LIN {X -0.262,Y -705.428,Z 1161.453,A 0.000,B 0.000,C 90.000,E1 117.462} C_DIS
LIN {X -0.017,Y -706.101,Z 1161.449,A 0.000,B 0.000,C 90.000,E1 116.744} C_DIS
LIN {X 0.213,Y -706.582,Z 1161.443,A 0.000,B 0.000,C 90.000,E1 115.796} C_DIS
LIN {X 0.157,Y -706.745,Z 1161.440,A 0.000,B 0.000,C 90.000,E1 115.103} C_DIS
LIN {X 0.105,Y -706.466,Z 1161.437,A 0.000,B 0.000,C 90.000,E1 114.643} C_DIS
LIN {X 0.398,Y -706.184,Z 1161.436,A 0.000,B 0.000,C 90.000,E1 114.387} C_DIS
LIN {X 0.046,Y -705.311,Z 1161.433,A 0.000,B 0.000,C 90.000,E1 113.951} C_DIS
LIN {X -0.310,Y -703.330,Z 1161.431,A 0.000,B 0.000,C 90.000,E1 113.515} C_DIS
LIN {X -0.028,Y -702.160,Z 1161.429,A 0.000,B 0.000,C 90.000,E1 113.259} C_DIS
LIN {X -0.027,Y -700.058,Z 1161.428,A 0.000,B 0.000,C 90.000,E1 113.025} C_DIS
LIN {X 0.371,Y -696.559,Z 1161.426,A 0.000,B 0.000,C 90.000,E1 112.642} C_DIS
LIN {X -0.143,Y -694.698,Z 1161.425,A 0.000,B 0.000,C 90.000,E1 112.567} C_DIS
LIN {X -0.188,Y -689.270,Z 1161.424,A 0.000,B 0.000,C 90.000,E1 112.386} C_DIS
LIN {X -0.184,Y -686.002,Z 1161.424,A 0.000,B 0.000,C 90.000,E1 112.280} C_DIS
LIN {X -0.175,Y -685.095,Z 1161.424,A 0.000,B 0.000,C 90.000,E1 112.259} C_DIS
LIN {X 0.074,Y -681.362,Z 1161.423,A 0.000,B 0.000,C 90.000,E1 112.206} C_DIS
LIN {X -0.288,Y -676.379,Z 1161.423,A 0.000,B 0.000,C 90.000,E1 112.206} C_DIS
LIN {X 0.256,Y -604.263,Z 1161.423,A 0.000,B 0.000,C 90.000,E1 112.153} C_DIS
LIN {X -0.142,Y -600.886,Z 1161.422,A 0.000,B 0.000,C 90.000,E1 111.972} C_DIS
LIN {X 0.084,Y -595.436,Z 1161.420,A 0.000,B 0.000,C 90.000,E1 111.535} C_DIS
LIN {X -0.058,Y -578.311,Z 1161.411,A 0.000,B 0.000,C 90.000,E1 110.066} C_DIS
LIN {X -0.053,Y -574.045,Z 1161.410,A 0.000,B 0.000,C 90.000,E1 109.704} C_DIS
LIN {X -0.238,Y -568.064,Z 1161.407,A 0.000,B 0.000,C 90.000,E1 109.268} C_DIS
LIN {X -0.148,Y -560.191,Z 1161.404,A 0.000,B 0.000,C 90.000,E1 108.725} C_DIS
LIN {X -0.132,Y -555.536,Z 1161.402,A 0.000,B 0.000,C 90.000,E1 108.417} C_DIS
LIN {X -0.186,Y -551.660,Z 1161.401,A 0.000,B 0.000,C 90.000,E1 108.109} C_DIS
LIN {X 0.019,Y -550.319,Z 1161.399,A 0.000,B 0.000,C 90.000,E1 107.873} C_DIS
LIN {X -0.023,Y -550.302,Z 1161.399,A 0.000,B 0.000,C 90.000,E1 107.873} C_DIS
LIN {X -0.264,Y -550.002,Z 1161.398,A 0.000,B 0.000,C 90.000,E1 107.583} C_DIS
LIN {X -0.119,Y -550.184,Z 1161.394,A 0.000,B 0.000,C 90.000,E1 106.968} C_DIS
LIN {X 0.015,Y -551.315,Z 1161.386,A 0.000,B 0.000,C 90.000,E1 105.552} C_DIS
LIN {X 0.018,Y -552.901,Z 1161.376,A 0.000,B 0.000,C 90.000,E1 103.592} C_DIS
LIN {X -0.071,Y -554.962,Z 1161.363,A 0.000,B 0.000,C 90.000,E1 101.366} C_DIS
LIN {X -0.095,Y -556.105,Z 1161.357,A 0.000,B 0.000,C 90.000,E1 100.254} C_DIS
LIN {X 0.066,Y -557.646,Z 1161.348,A 0.000,B 0.000,C 90.000,E1 98.568} C_DIS
LIN {X 0.038,Y -558.878,Z 1161.340,A 0.000,B 0.000,C 90.000,E1 97.182} C_DIS
LIN {X 0.244,Y -560.316,Z 1161.329,A 0.000,B 0.000,C 90.000,E1 95.220} C_DIS
LIN {X -0.267,Y -561.478,Z 1161.320,A 0.000,B 0.000,C 90.000,E1 93.612} C_DIS
LIN {X -0.219,Y -562.750,Z 1161.311,A 0.000,B 0.000,C 90.000,E1 91.949} C_DIS
LIN {X -0.250,Y -563.791,Z 1161.303,A 0.000,B 0.000,C 90.000,E1 90.573} C_DIS
LIN {X 0.180,Y -564.631,Z 1161.297,A 0.000,B 0.000,C 90.000,E1 89.427} C_DIS
LIN {X -0.271,Y -565.665,Z 1161.288,A 0.000,B 0.000,C 90.000,E1 87.822} C_DIS
LIN {X -0.139,Y -566.641,Z 1161.279,A 0.000,B 0.000,C 90.000,E1 86.159} C_DIS
LIN {X 0.200,Y -567.813,Z 1161.268,A 0.000,B 0.000,C 90.000,E1 84.204} C_DIS
LIN {X -0.212,Y -568.704,Z 1161.260,A 0.000,B 0.000,C 90.000,E1 82.875} C_DIS
LIN {X -0.043,Y -569.488,Z 1161.253,A 0.000,B 0.000,C 90.000,E1 81.489} C_DIS
LIN {X 0.221,Y -570.126,Z 1161.245,A 0.000,B 0.000,C 90.000,E1 80.095} C_DIS
LIN {X 0.122,Y -570.936,Z 1161.236,A 0.000,B 0.000,C 90.000,E1 78.465} C_DIS
LIN {X -0.235,Y -571.445,Z 1161.230,A 0.000,B 0.000,C 90.000,E1 77.409} C_DIS
LIN {X 0.126,Y -572.386,Z 1161.219,A 0.000,B 0.000,C 90.000,E1 75.463} C_DIS
LIN {X -0.259,Y -573.550,Z 1161.207,A 0.000,B 0.000,C 90.000,E1 73.323} C_DIS
LIN {X -0.089,Y -574.421,Z 1161.200,A 0.000,B 0.000,C 90.000,E1 71.945} C_DIS
LIN {X -0.261,Y -576.180,Z 1161.186,A 0.000,B 0.000,C 90.000,E1 69.518} C_DIS
LIN {X -0.193,Y -577.810,Z 1161.176,A 0.000,B 0.000,C 90.000,E1 67.614} C_DIS
LIN {X -0.021,Y -579.444,Z 1161.167,A 0.000,B 0.000,C 90.000,E1 65.973} C_DIS
LIN {X 0.198,Y -580.890,Z 1161.158,A 0.000,B 0.000,C 90.000,E1 64.332} C_DIS
LIN {X -0.215,Y -582.678,Z 1161.147,A 0.000,B 0.000,C 90.000,E1 62.487} C_DIS
LIN {X -0.077,Y -583.908,Z 1161.140,A 0.000,B 0.000,C 90.000,E1 61.129} C_DIS
LIN {X -0.143,Y -585.014,Z 1161.132,A 0.000,B 0.000,C 90.000,E1 59.793} C_DIS
LIN {X -0.357,Y -585.879,Z 1161.126,A 0.000,B 0.000,C 90.000,E1 58.742} C_DIS
LIN {X -0.209,Y -586.962,Z 1161.117,A 0.000,B 0.000,C 90.000,E1 57.120} C_DIS
LIN {X 0.225,Y -587.735,Z 1161.111,A 0.000,B 0.000,C 90.000,E1 56.008} C_DIS
LIN {X 0.251,Y -588.690,Z 1161.102,A 0.000,B 0.000,C 90.000,E1 54.402} C_DIS
LIN {X 0.020,Y -589.819,Z 1161.092,A 0.000,B 0.000,C 90.000,E1 52.557} C_DIS
LIN {X -0.249,Y -590.539,Z 1161.085,A 0.000,B 0.000,C 90.000,E1 51.251} C_DIS
LIN {X 0.115,Y -591.104,Z 1161.079,A 0.000,B 0.000,C 90.000,E1 50.150} C_DIS
LIN {X -0.174,Y -591.386,Z 1161.074,A 0.000,B 0.000,C 90.000,E1 49.380} C_DIS
LIN {X 0.104,Y -591.737,Z 1161.065,A 0.000,B 0.000,C 90.000,E1 47.757} C_DIS
LIN {X -0.213,Y -591.813,Z 1161.058,A 0.000,B 0.000,C 90.000,E1 46.458} C_DIS
LIN {X -0.319,Y -591.679,Z 1161.052,A 0.000,B 0.000,C 90.000,E1 45.405} C_DIS
LIN {X 0.047,Y -591.602,Z 1161.049,A 0.000,B 0.000,C 90.000,E1 44.838} C_DIS
LIN {X -0.062,Y -591.163,Z 1161.043,A 0.000,B 0.000,C 90.000,E1 43.785} C_DIS
LIN {X 0.009,Y -590.467,Z 1161.036,A 0.000,B 0.000,C 90.000,E1 42.447} C_DIS
LIN {X -0.086,Y -589.582,Z 1161.030,A 0.000,B 0.000,C 90.000,E1 41.391} C_DIS
LIN {X 0.010,Y -588.204,Z 1161.023,A 0.000,B 0.000,C 90.000,E1 40.048} C_DIS
LIN {X -0.304,Y -587.257,Z 1161.018,A 0.000,B 0.000,C 90.000,E1 39.277} C_DIS
LIN {X 0.203,Y -585.495,Z 1161.011,A 0.000,B 0.000,C 90.000,E1 37.890} C_DIS
LIN {X -0.328,Y -583.805,Z 1161.005,A 0.000,B 0.000,C 90.000,E1 36.870} C_DIS
LIN {X 0.055,Y -581.695,Z 1160.999,A 0.000,B 0.000,C 90.000,E1 35.758} C_DIS
LIN {X 0.102,Y -579.797,Z 1160.994,A 0.000,B 0.000,C 90.000,E1 34.945} C_DIS
LIN {X 0.264,Y -577.702,Z 1160.990,A 0.000,B 0.000,C 90.000,E1 34.119} C_DIS
LIN {X -0.392,Y -575.196,Z 1160.985,A 0.000,B 0.000,C 90.000,E1 33.372} C_DIS
LIN {X -0.102,Y -573.425,Z 1160.982,A 0.000,B 0.000,C 90.000,E1 32.801} C_DIS
LIN {X 0.295,Y -569.267,Z 1160.976,A 0.000,B 0.000,C 90.000,E1 31.671} C_DIS
LIN {X 0.047,Y -565.634,Z 1160.972,A 0.000,B 0.000,C 90.000,E1 30.875} C_DIS
LIN {X -0.141,Y -562.314,Z 1160.968,A 0.000,B 0.000,C 90.000,E1 30.207} C_DIS
LIN {X 0.195,Y -557.244,Z 1160.962,A 0.000,B 0.000,C 90.000,E1 29.205} C_DIS
LIN {X -0.076,Y -553.266,Z 1160.958,A 0.000,B 0.000,C 90.000,E1 28.537} C_DIS
LIN {X -0.039,Y -549.883,Z 1160.955,A 0.000,B 0.000,C 90.000,E1 27.975} C_DIS
LIN {X 0.231,Y -546.282,Z 1160.952,A 0.000,B 0.000,C 90.000,E1 27.385} C_DIS
LIN {X -0.134,Y -543.457,Z 1160.950,A 0.000,B 0.000,C 90.000,E1 27.001} C_DIS
LIN {X -0.047,Y -538.223,Z 1160.946,A 0.000,B 0.000,C 90.000,E1 26.283} C_DIS
LIN {X -0.107,Y -533.817,Z 1160.943,A 0.000,B 0.000,C 90.000,E1 25.720} C_DIS
LIN {X -0.008,Y -526.846,Z 1160.938,A 0.000,B 0.000,C 90.000,E1 24.847} C_DIS
LIN {X -0.137,Y -519.286,Z 1160.933,A 0.000,B 0.000,C 90.000,E1 24.003} C_DIS
LIN {X 0.240,Y -512.837,Z 1160.929,A 0.000,B 0.000,C 90.000,E1 23.259} C_DIS
LIN {X -0.093,Y -505.969,Z 1160.926,A 0.000,B 0.000,C 90.000,E1 22.589} C_DIS
LIN {X 0.046,Y -500.450,Z 1160.922,A 0.000,B 0.000,C 90.000,E1 22.025} C_DIS
LIN {X -0.062,Y -490.576,Z 1160.917,A 0.000,B 0.000,C 90.000,E1 21.099} C_DIS
LIN {X -0.006,Y -480.430,Z 1160.912,A 0.000,B 0.000,C 90.000,E1 20.174} C_DIS
LIN {X -0.115,Y -467.433,Z 1160.906,A 0.000,B 0.000,C 90.000,E1 19.014} C_DIS
LIN {X 0.017,Y -442.601,Z 1160.893,A 0.000,B 0.000,C 90.000,E1 16.732} C_DIS
LIN {X 0.098,Y -429.624,Z 1160.886,A 0.000,B 0.000,C 90.000,E1 15.426} C_DIS
LIN {X -0.121,Y -416.956,Z 1160.878,A 0.000,B 0.000,C 90.000,E1 14.064} C_DIS
LIN {X -0.221,Y -406.260,Z 1160.871,A 0.000,B 0.000,C 90.000,E1 12.771} C_DIS
LIN {X 0.195,Y -397.899,Z 1160.864,A 0.000,B 0.000,C 90.000,E1 11.535} C_DIS
LIN {X -0.133,Y -395.271,Z 1160.862,A 0.000,B 0.000,C 90.000,E1 11.130} C_DIS
LIN {X 0.077,Y -393.627,Z 1160.860,A 0.000,B 0.000,C 90.000,E1 10.715} C_DIS
LIN {X 0.022,Y -392.924,Z 1160.859,A 0.000,B 0.000,C 90.000,E1 10.546} C_DIS
LIN {X -0.016,Y -392.907,Z 1160.859,A 0.000,B 0.000,C 90.000,E1 10.546} C_DIS
LIN {X 0.149,Y -392.617,Z 1160.856,A 0.000,B 0.000,C 90.000,E1 10.084} C_DIS
LIN {X -0.047,Y -393.292,Z 1160.854,A 0.000,B 0.000,C 90.000,E1 9.670} C_DIS
LIN {X -0.129,Y -395.148,Z 1160.850,A 0.000,B 0.000,C 90.000,E1 8.973} C_DIS
LIN {X 0.162,Y -398.575,Z 1160.844,A 0.000,B 0.000,C 90.000,E1 7.871} C_DIS
LIN {X -0.086,Y -401.754,Z 1160.839,A 0.000,B 0.000,C 90.000,E1 7.068} C_DIS
LIN {X -0.104,Y -405.686,Z 1160.835,A 0.000,B 0.000,C 90.000,E1 6.372} C_DIS
LIN {X -0.128,Y -406.747,Z 1160.834,A 0.000,B 0.000,C 90.000,E1 6.201} C_DIS
LIN {X 0.009,Y -407.934,Z 1160.834,A 0.000,B 0.000,C 90.000,E1 6.030} C_DIS
LIN {X -0.107,Y -410.829,Z 1160.832,A 0.000,B 0.000,C 90.000,E1 5.739} C_DIS
LIN {X -0.033,Y -414.950,Z 1160.830,A 0.000,B 0.000,C 90.000,E1 5.391} C_DIS
LIN {X -0.070,Y -429.560,Z 1160.824,A 0.000,B 0.000,C 90.000,E1 4.302} C_DIS
LIN {X -0.226,Y -444.055,Z 1160.818,A 0.000,B 0.000,C 90.000,E1 3.269} C_DIS
LIN {X 0.022,Y -465.153,Z 1160.810,A 0.000,B 0.000,C 90.000,E1 1.776} C_DIS
LIN {X -0.135,Y -476.141,Z 1160.806,A 0.000,B 0.000,C 90.000,E1 1.031} C_DIS
LIN {X -0.094,Y -483.837,Z 1160.802,A 0.000,B 0.000,C 90.000,E1 0.458} C_DIS
LIN {X 0.000,Y -489.788,Z 1160.800,A 0.000,B 0.000,C 90.000,E1 360.000} C_DIS
LIN {X -0.023,Y -496.862,Z 1160.797,A 0.000,B 0.000,C 90.000,E1 359.427} C_DIS
LIN {X -0.096,Y -504.041,Z 1160.793,A 0.000,B 0.000,C 90.000,E1 358.797} C_DIS
LIN {X 0.239,Y -509.609,Z 1160.790,A 0.000,B 0.000,C 90.000,E1 358.224} C_DIS
LIN {X -0.168,Y -516.066,Z 1160.787,A 0.000,B 0.000,C 90.000,E1 357.593} C_DIS
LIN {X 0.067,Y -522.425,Z 1160.783,A 0.000,B 0.000,C 90.000,E1 356.846} C_DIS
LIN {X 0.244,Y -528.292,Z 1160.779,A 0.000,B 0.000,C 90.000,E1 356.102} C_DIS
LIN {X 0.224,Y -532.626,Z 1160.775,A 0.000,B 0.000,C 90.000,E1 355.527} C_DIS
LIN {X -0.036,Y -537.342,Z 1160.771,A 0.000,B 0.000,C 90.000,E1 354.837} C_DIS
LIN {X -0.257,Y -541.657,Z 1160.767,A 0.000,B 0.000,C 90.000,E1 354.147} C_DIS
LIN {X 0.158,Y -545.578,Z 1160.763,A 0.000,B 0.000,C 90.000,E1 353.394} C_DIS
LIN {X 0.267,Y -548.451,Z 1160.760,A 0.000,B 0.000,C 90.000,E1 352.818} C_DIS
LIN {X 0.247,Y -552.943,Z 1160.755,A 0.000,B 0.000,C 90.000,E1 351.837} C_DIS
LIN {X 0.229,Y -555.790,Z 1160.751,A 0.000,B 0.000,C 90.000,E1 351.141} C_DIS
LIN {X -0.017,Y -558.814,Z 1160.746,A 0.000,B 0.000,C 90.000,E1 350.330} C_DIS
LIN {X -0.137,Y -561.551,Z 1160.742,A 0.000,B 0.000,C 90.000,E1 349.511} C_DIS
LIN {X 0.219,Y -564.082,Z 1160.737,A 0.000,B 0.000,C 90.000,E1 348.645} C_DIS
LIN {X -0.058,Y -567.941,Z 1160.729,A 0.000,B 0.000,C 90.000,E1 347.297} C_DIS
LIN {X -0.139,Y -571.408,Z 1160.722,A 0.000,B 0.000,C 90.000,E1 345.936} C_DIS
LIN {X 0.208,Y -574.072,Z 1160.716,A 0.000,B 0.000,C 90.000,E1 344.810} C_DIS
LIN {X -0.316,Y -577.142,Z 1160.708,A 0.000,B 0.000,C 90.000,E1 343.504} C_DIS
LIN {X 0.307,Y -580.713,Z 1160.699,A 0.000,B 0.000,C 90.000,E1 341.819} C_DIS
LIN {X 0.003,Y -582.324,Z 1160.695,A 0.000,B 0.000,C 90.000,E1 341.040} C_DIS
LIN {X 0.310,Y -584.331,Z 1160.689,A 0.000,B 0.000,C 90.000,E1 339.934} C_DIS
LIN {X 0.312,Y -586.470,Z 1160.681,A 0.000,B 0.000,C 90.000,E1 338.592} C_DIS
LIN {X -0.160,Y -587.244,Z 1160.678,A 0.000,B 0.000,C 90.000,E1 338.103} C_DIS
LIN {X 0.097,Y -588.618,Z 1160.671,A 0.000,B 0.000,C 90.000,E1 336.741} C_DIS
LIN {X 0.294,Y -589.141,Z 1160.666,A 0.000,B 0.000,C 90.000,E1 335.921} C_DIS
LIN {X -0.034,Y -589.396,Z 1160.662,A 0.000,B 0.000,C 90.000,E1 335.153} C_DIS
LIN {X 0.178,Y -589.369,Z 1160.658,A 0.000,B 0.000,C 90.000,E1 334.332} C_DIS
LIN {X -0.142,Y -589.023,Z 1160.653,A 0.000,B 0.000,C 90.000,E1 333.563} C_DIS
LIN {X 0.059,Y -588.261,Z 1160.649,A 0.000,B 0.000,C 90.000,E1 332.743} C_DIS
LIN {X -0.163,Y -587.616,Z 1160.646,A 0.000,B 0.000,C 90.000,E1 332.231} C_DIS
LIN {X -0.228,Y -586.211,Z 1160.641,A 0.000,B 0.000,C 90.000,E1 331.435} C_DIS
LIN {X 0.209,Y -584.479,Z 1160.637,A 0.000,B 0.000,C 90.000,E1 330.589} C_DIS
LIN {X 0.118,Y -582.277,Z 1160.632,A 0.000,B 0.000,C 90.000,E1 329.793} C_DIS
LIN {X 0.004,Y -579.589,Z 1160.628,A 0.000,B 0.000,C 90.000,E1 328.997} C_DIS
LIN {X -0.063,Y -576.929,Z 1160.624,A 0.000,B 0.000,C 90.000,E1 328.329} C_DIS
LIN {X 0.064,Y -572.768,Z 1160.620,A 0.000,B 0.000,C 90.000,E1 327.502} C_DIS
LIN {X 0.023,Y -569.600,Z 1160.617,A 0.000,B 0.000,C 90.000,E1 326.962} C_DIS
LIN {X 0.073,Y -564.104,Z 1160.612,A 0.000,B 0.000,C 90.000,E1 326.135} C_DIS
LIN {X -0.031,Y -560.179,Z 1160.609,A 0.000,B 0.000,C 90.000,E1 325.595} C_DIS
LIN {X -0.050,Y -556.903,Z 1160.607,A 0.000,B 0.000,C 90.000,E1 325.182} C_DIS
LIN {X 0.137,Y -551.314,Z 1160.603,A 0.000,B 0.000,C 90.000,E1 324.482} C_DIS
LIN {X 0.302,Y -543.898,Z 1160.598,A 0.000,B 0.000,C 90.000,E1 323.623} C_DIS
LIN {X -0.197,Y -536.207,Z 1160.594,A 0.000,B 0.000,C 90.000,E1 322.844} C_DIS
LIN {X 0.016,Y -529.985,Z 1160.590,A 0.000,B 0.000,C 90.000,E1 322.145} C_DIS
LIN {X 0.327,Y -527.584,Z 1160.588,A 0.000,B 0.000,C 90.000,E1 321.823} C_DIS
LIN {X 0.268,Y -524.788,Z 1160.586,A 0.000,B 0.000,C 90.000,E1 321.457} C_DIS
LIN {X 0.044,Y -522.012,Z 1160.583,A 0.000,B 0.000,C 90.000,E1 321.009} C_DIS
LIN {X -0.141,Y -521.321,Z 1160.583,A 0.000,B 0.000,C 90.000,E1 320.884} C_DIS
LIN {X -0.227,Y -519.739,Z 1160.580,A 0.000,B 0.000,C 90.000,E1 320.436} C_DIS
LIN {X 0.132,Y -518.543,Z 1160.576,A 0.000,B 0.000,C 90.000,E1 319.666} C_DIS
LIN {X -0.033,Y -518.632,Z 1160.569,A 0.000,B 0.000,C 90.000,E1 318.366} C_DIS
LIN {X -0.127,Y -519.406,Z 1160.559,A 0.000,B 0.000,C 90.000,E1 316.620} C_DIS
LIN {X 0.045,Y -520.418,Z 1160.548,A 0.000,B 0.000,C 90.000,E1 314.555} C_DIS
LIN {X -0.051,Y -521.275,Z 1160.538,A 0.000,B 0.000,C 90.000,E1 312.813} C_DIS
LIN {X -0.143,Y -522.416,Z 1160.526,A 0.000,B 0.000,C 90.000,E1 310.782} C_DIS
LIN {X -0.197,Y -523.548,Z 1160.515,A 0.000,B 0.000,C 90.000,E1 308.749} C_DIS
LIN {X -0.116,Y -524.617,Z 1160.505,A 0.000,B 0.000,C 90.000,E1 306.996} C_DIS
LIN {X 0.162,Y -525.317,Z 1160.499,A 0.000,B 0.000,C 90.000,E1 305.804} C_DIS
LIN {X -0.311,Y -526.137,Z 1160.491,A 0.000,B 0.000,C 90.000,E1 304.405} C_DIS
LIN {X 0.002,Y -527.633,Z 1160.478,A 0.000,B 0.000,C 90.000,E1 302.054} C_DIS
LIN {X -0.142,Y -528.689,Z 1160.469,A 0.000,B 0.000,C 90.000,E1 300.335} C_DIS
LIN {X -0.070,Y -529.202,Z 1160.464,A 0.000,B 0.000,C 90.000,E1 299.461} C_DIS
LIN {X -0.090,Y -529.711,Z 1160.457,A 0.000,B 0.000,C 90.000,E1 298.309} C_DIS
LIN {X -0.021,Y -530.066,Z 1160.453,A 0.000,B 0.000,C 90.000,E1 297.436} C_DIS
LIN {X -0.142,Y -530.367,Z 1160.443,A 0.000,B 0.000,C 90.000,E1 295.720} C_DIS
LIN {X 0.041,Y -530.419,Z 1160.435,A 0.000,B 0.000,C 90.000,E1 294.259} C_DIS
LIN {X -0.113,Y -530.369,Z 1160.424,A 0.000,B 0.000,C 90.000,E1 292.259} C_DIS
LIN {X 0.138,Y -530.298,Z 1160.416,A 0.000,B 0.000,C 90.000,E1 290.791} C_DIS
LIN {X -0.101,Y -529.831,Z 1160.406,A 0.000,B 0.000,C 90.000,E1 289.087} C_DIS
LIN {X -0.210,Y -529.453,Z 1160.400,A 0.000,B 0.000,C 90.000,E1 287.946} C_DIS
LIN {X -0.128,Y -528.736,Z 1160.390,A 0.000,B 0.000,C 90.000,E1 286.205} C_DIS
LIN {X 0.088,Y -528.396,Z 1160.385,A 0.000,B 0.000,C 90.000,E1 285.315} C_DIS
LIN {X -0.006,Y -527.467,Z 1160.376,A 0.000,B 0.000,C 90.000,E1 283.592} C_DIS
LIN {X 0.210,Y -526.778,Z 1160.369,A 0.000,B 0.000,C 90.000,E1 282.411} C_DIS
LIN {X -0.195,Y -525.859,Z 1160.361,A 0.000,B 0.000,C 90.000,E1 281.007} C_DIS
LIN {X -0.193,Y -524.860,Z 1160.353,A 0.000,B 0.000,C 90.000,E1 279.557} C_DIS
LIN {X -0.195,Y -523.779,Z 1160.343,A 0.000,B 0.000,C 90.000,E1 277.814} C_DIS
LIN {X 0.161,Y -522.723,Z 1160.334,A 0.000,B 0.000,C 90.000,E1 276.030} C_DIS
LIN {X -0.017,Y -521.895,Z 1160.324,A 0.000,B 0.000,C 90.000,E1 274.302} C_DIS
LIN {X -0.209,Y -521.260,Z 1160.316,A 0.000,B 0.000,C 90.000,E1 272.865} C_DIS
LIN {X 0.077,Y -520.691,Z 1160.308,A 0.000,B 0.000,C 90.000,E1 271.375} C_DIS
LIN {X -0.178,Y -520.061,Z 1160.300,A 0.000,B 0.000,C 90.000,E1 269.943} C_DIS
LIN {X 0.074,Y -519.452,Z 1160.292,A 0.000,B 0.000,C 90.000,E1 268.453} C_DIS
LIN {X -0.195,Y -518.750,Z 1160.283,A 0.000,B 0.000,C 90.000,E1 267.020} C_DIS
LIN {X 0.072,Y -517.852,Z 1160.275,A 0.000,B 0.000,C 90.000,E1 265.527} C_DIS
LIN {X -0.194,Y -516.745,Z 1160.267,A 0.000,B 0.000,C 90.000,E1 264.090} C_DIS
LIN {X 0.058,Y -515.023,Z 1160.257,A 0.000,B 0.000,C 90.000,E1 262.299} C_DIS
LIN {X -0.158,Y -513.287,Z 1160.247,A 0.000,B 0.000,C 90.000,E1 260.557} C_DIS
LIN {X 0.060,Y -511.322,Z 1160.236,A 0.000,B 0.000,C 90.000,E1 258.465} C_DIS
LIN {X -0.118,Y -509.260,Z 1160.223,A 0.000,B 0.000,C 90.000,E1 256.117} C_DIS
LIN {X -0.053,Y -507.467,Z 1160.211,A 0.000,B 0.000,C 90.000,E1 254.031} C_DIS
LIN {X 0.033,Y -505.854,Z 1160.201,A 0.000,B 0.000,C 90.000,E1 252.236} C_DIS
LIN {X 0.231,Y -504.171,Z 1160.191,A 0.000,B 0.000,C 90.000,E1 250.423} C_DIS
LIN {X 0.168,Y -502.118,Z 1160.180,A 0.000,B 0.000,C 90.000,E1 248.337} C_DIS
LIN {X -0.177,Y -500.917,Z 1160.173,A 0.000,B 0.000,C 90.000,E1 247.177} C_DIS
LIN {X 0.236,Y -499.874,Z 1160.168,A 0.000,B 0.000,C 90.000,E1 246.230} C_DIS
LIN {X 0.314,Y -498.049,Z 1160.160,A 0.000,B 0.000,C 90.000,E1 244.717} C_DIS
LIN {X -0.095,Y -496.048,Z 1160.151,A 0.000,B 0.000,C 90.000,E1 243.256} C_DIS
LIN {X 0.118,Y -493.945,Z 1160.143,A 0.000,B 0.000,C 90.000,E1 241.719} C_DIS
LIN {X -0.083,Y -491.277,Z 1160.133,A 0.000,B 0.000,C 90.000,E1 239.921} C_DIS
LIN {X 0.261,Y -489.514,Z 1160.126,A 0.000,B 0.000,C 90.000,E1 238.663} C_DIS
LIN {X -0.014,Y -487.185,Z 1160.118,A 0.000,B 0.000,C 90.000,E1 237.168} C_DIS
LIN {X -0.061,Y -484.884,Z 1160.109,A 0.000,B 0.000,C 90.000,E1 235.642} C_DIS
LIN {X 0.056,Y -482.159,Z 1160.099,A 0.000,B 0.000,C 90.000,E1 233.783} C_DIS
LIN {X -0.012,Y -480.267,Z 1160.092,A 0.000,B 0.000,C 90.000,E1 232.557} C_DIS
LIN {X 0.061,Y -476.440,Z 1160.078,A 0.000,B 0.000,C 90.000,E1 230.070} C_DIS
LIN {X -0.060,Y -474.104,Z 1160.070,A 0.000,B 0.000,C 90.000,E1 228.528} C_DIS
LIN {X 0.126,Y -471.588,Z 1160.061,A 0.000,B 0.000,C 90.000,E1 226.944} C_DIS
LIN {X 0.098,Y -465.961,Z 1160.040,A 0.000,B 0.000,C 90.000,E1 223.176} C_DIS
LIN {X 0.002,Y -462.302,Z 1160.017,A 0.000,B 0.000,C 90.000,E1 219.072} C_DIS
LIN {X -0.181,Y -461.000,Z 1160.005,A 0.000,B 0.000,C 90.000,E1 216.870} C_DIS
LIN {X -0.011,Y -459.562,Z 1159.976,A 0.000,B 0.000,C 90.000,E1 211.750} C_DIS
LIN {X 0.092,Y -460.857,Z 1159.957,A 0.000,B 0.000,C 90.000,E1 208.231} C_DIS
LIN {X -0.214,Y -462.289,Z 1159.946,A 0.000,B 0.000,C 90.000,E1 206.360} C_DIS
LIN {X 0.205,Y -465.295,Z 1159.932,A 0.000,B 0.000,C 90.000,E1 203.770} C_DIS
LIN {X 0.224,Y -471.462,Z 1159.913,A 0.000,B 0.000,C 90.000,E1 200.301} C_DIS
LIN {X 0.082,Y -477.505,Z 1159.899,A 0.000,B 0.000,C 90.000,E1 197.819} C_DIS
LIN {X -0.155,Y -484.717,Z 1159.885,A 0.000,B 0.000,C 90.000,E1 195.371} C_DIS
LIN {X -0.197,Y -490.749,Z 1159.875,A 0.000,B 0.000,C 90.000,E1 193.536} C_DIS
LIN {X -0.127,Y -495.808,Z 1159.867,A 0.000,B 0.000,C 90.000,E1 192.007} C_DIS
LIN {X -0.134,Y -502.173,Z 1159.857,A 0.000,B 0.000,C 90.000,E1 190.197} C_DIS
LIN {X -0.183,Y -510.885,Z 1159.843,A 0.000,B 0.000,C 90.000,E1 187.814} C_DIS
LIN {X 0.008,Y -516.405,Z 1159.835,A 0.000,B 0.000,C 90.000,E1 186.315} C_DIS
LIN {X 0.244,Y -522.816,Z 1159.825,A 0.000,B 0.000,C 90.000,E1 184.531} C_DIS
LIN {X 0.095,Y -527.125,Z 1159.819,A 0.000,B 0.000,C 90.000,E1 183.383} C_DIS
LIN {X -0.006,Y -532.466,Z 1159.811,A 0.000,B 0.000,C 90.000,E1 181.949} C_DIS
LIN {X -0.015,Y -537.760,Z 1159.803,A 0.000,B 0.000,C 90.000,E1 180.516} C_DIS
LIN {X 0.087,Y -544.151,Z 1159.793,A 0.000,B 0.000,C 90.000,E1 178.797} C_DIS
LIN {X -0.211,Y -550.558,Z 1159.784,A 0.000,B 0.000,C 90.000,E1 177.135} C_DIS
LIN {X -0.234,Y -557.962,Z 1159.773,A 0.000,B 0.000,C 90.000,E1 175.179} C_DIS
LIN {X 0.260,Y -563.175,Z 1159.765,A 0.000,B 0.000,C 90.000,E1 173.742} C_DIS
LIN {X -0.120,Y -569.471,Z 1159.756,A 0.000,B 0.000,C 90.000,E1 172.129} C_DIS
LIN {X -0.211,Y -575.692,Z 1159.747,A 0.000,B 0.000,C 90.000,E1 170.500} C_DIS
LIN {X -0.163,Y -581.770,Z 1159.738,A 0.000,B 0.000,C 90.000,E1 168.870} C_DIS
LIN {X 0.207,Y -585.764,Z 1159.732,A 0.000,B 0.000,C 90.000,E1 167.757} C_DIS
LIN {X -0.254,Y -590.583,Z 1159.725,A 0.000,B 0.000,C 90.000,E1 166.464} C_DIS
LIN {X 0.082,Y -595.199,Z 1159.717,A 0.000,B 0.000,C 90.000,E1 165.102} C_DIS
LIN {X 0.047,Y -598.842,Z 1159.711,A 0.000,B 0.000,C 90.000,E1 164.047} C_DIS
LIN {X -0.185,Y -602.353,Z 1159.706,A 0.000,B 0.000,C 90.000,E1 163.015} C_DIS
LIN {X -0.052,Y -606.543,Z 1159.698,A 0.000,B 0.000,C 90.000,E1 161.692} C_DIS
LIN {X 0.088,Y -611.258,Z 1159.690,A 0.000,B 0.000,C 90.000,E1 160.115} C_DIS
LIN {X -0.260,Y -615.792,Z 1159.681,A 0.000,B 0.000,C 90.000,E1 158.592} C_DIS
LIN {X -0.304,Y -620.038,Z 1159.672,A 0.000,B 0.000,C 90.000,E1 157.050} C_DIS
LIN {X -0.023,Y -623.514,Z 1159.665,A 0.000,B 0.000,C 90.000,E1 155.741} C_DIS
LIN {X 0.028,Y -627.493,Z 1159.657,A 0.000,B 0.000,C 90.000,E1 154.204} C_DIS
LIN {X 0.172,Y -631.334,Z 1159.648,A 0.000,B 0.000,C 90.000,E1 152.666} C_DIS
LIN {X 0.308,Y -633.801,Z 1159.643,A 0.000,B 0.000,C 90.000,E1 151.641} C_DIS
LIN {X -0.049,Y -636.689,Z 1159.636,A 0.000,B 0.000,C 90.000,E1 150.411} C_DIS
LIN {X -0.099,Y -638.966,Z 1159.630,A 0.000,B 0.000,C 90.000,E1 149.410} C_DIS
LIN {X -0.117,Y -641.027,Z 1159.625,A 0.000,B 0.000,C 90.000,E1 148.408} C_DIS
LIN {X 0.288,Y -643.463,Z 1159.618,A 0.000,B 0.000,C 90.000,E1 147.120} C_DIS
LIN {X 0.195,Y -645.797,Z 1159.611,A 0.000,B 0.000,C 90.000,E1 145.881} C_DIS
LIN {X 0.136,Y -647.982,Z 1159.604,A 0.000,B 0.000,C 90.000,E1 144.642} C_DIS
LIN {X -0.040,Y -650.110,Z 1159.597,A 0.000,B 0.000,C 90.000,E1 143.417} C_DIS
LIN {X -0.260,Y -653.420,Z 1159.586,A 0.000,B 0.000,C 90.000,E1 141.457} C_DIS
LIN {X 0.016,Y -657.097,Z 1159.575,A 0.000,B 0.000,C 90.000,E1 139.461} C_DIS
LIN {X -0.147,Y -660.626,Z 1159.565,A 0.000,B 0.000,C 90.000,E1 137.757} C_DIS
LIN {X -0.219,Y -663.632,Z 1159.557,A 0.000,B 0.000,C 90.000,E1 136.296} C_DIS
LIN {X -0.253,Y -668.791,Z 1159.544,A 0.000,B 0.000,C 90.000,E1 133.866} C_DIS
LIN {X -0.133,Y -673.295,Z 1159.533,A 0.000,B 0.000,C 90.000,E1 131.919} C_DIS
LIN {X 0.197,Y -678.478,Z 1159.521,A 0.000,B 0.000,C 90.000,E1 129.725} C_DIS
LIN {X 0.002,Y -681.542,Z 1159.514,A 0.000,B 0.000,C 90.000,E1 128.543} C_DIS
LIN {X -0.151,Y -684.520,Z 1159.508,A 0.000,B 0.000,C 90.000,E1 127.363} C_DIS
LIN {X -0.126,Y -687.507,Z 1159.501,A 0.000,B 0.000,C 90.000,E1 126.171} C_DIS
LIN {X -0.011,Y -691.004,Z 1159.493,A 0.000,B 0.000,C 90.000,E1 124.739} C_DIS
LIN {X 0.086,Y -693.272,Z 1159.488,A 0.000,B 0.000,C 90.000,E1 123.785} C_DIS
LIN {X -0.105,Y -696.493,Z 1159.480,A 0.000,B 0.000,C 90.000,E1 122.388} C_DIS
LIN {X 0.035,Y -697.969,Z 1159.476,A 0.000,B 0.000,C 90.000,E1 121.671} C_DIS
LIN {X -0.121,Y -700.212,Z 1159.469,A 0.000,B 0.000,C 90.000,E1 120.512} C_DIS
LIN {X 0.274,Y -702.683,Z 1159.462,A 0.000,B 0.000,C 90.000,E1 119.077} C_DIS
LIN {X 0.157,Y -704.340,Z 1159.457,A 0.000,B 0.000,C 90.000,E1 118.153} C_DIS
LIN {X 0.064,Y -705.376,Z 1159.453,A 0.000,B 0.000,C 90.000,E1 117.462} C_DIS
LIN {X 0.308,Y -706.055,Z 1159.449,A 0.000,B 0.000,C 90.000,E1 116.744} C_DIS
LIN {X -0.099,Y -706.543,Z 1159.444,A 0.000,B 0.000,C 90.000,E1 115.848} C_DIS
LIN {X -0.158,Y -706.735,Z 1159.440,A 0.000,B 0.000,C 90.000,E1 115.155} C_DIS
LIN {X -0.212,Y -706.481,Z 1159.437,A 0.000,B 0.000,C 90.000,E1 114.695} C_DIS
LIN {X -0.213,Y -706.228,Z 1159.436,A 0.000,B 0.000,C 90.000,E1 114.463} C_DIS
LIN {X 0.370,Y -705.358,Z 1159.433,A 0.000,B 0.000,C 90.000,E1 113.951} C_DIS
LIN {X -0.273,Y -704.507,Z 1159.432,A 0.000,B 0.000,C 90.000,E1 113.770} C_DIS
LIN {X 0.295,Y -702.331,Z 1159.429,A 0.000,B 0.000,C 90.000,E1 113.259} C_DIS
LIN {X 0.157,Y -701.438,Z 1159.429,A 0.000,B 0.000,C 90.000,E1 113.153} C_DIS
LIN {X 0.050,Y -696.897,Z 1159.426,A 0.000,B 0.000,C 90.000,E1 112.695} C_DIS
LIN {X -0.088,Y -695.236,Z 1159.426,A 0.000,B 0.000,C 90.000,E1 112.589} C_DIS
LIN {X 0.264,Y -692.820,Z 1159.425,A 0.000,B 0.000,C 90.000,E1 112.461} C_DIS
LIN {X -0.081,Y -685.622,Z 1159.424,A 0.000,B 0.000,C 90.000,E1 112.259} C_DIS
LIN {X 0.167,Y -683.209,Z 1159.423,A 0.000,B 0.000,C 90.000,E1 112.206} C_DIS
LIN {X -0.303,Y -677.072,Z 1159.423,A 0.000,B 0.000,C 90.000,E1 112.206} C_DIS
LIN {X 0.242,Y -604.198,Z 1159.423,A 0.000,B 0.000,C 90.000,E1 112.153} C_DIS
LIN {X -0.070,Y -600.945,Z 1159.422,A 0.000,B 0.000,C 90.000,E1 111.972} C_DIS
LIN {X 0.156,Y -595.490,Z 1159.420,A 0.000,B 0.000,C 90.000,E1 111.535} C_DIS
LIN {X 0.108,Y -578.472,Z 1159.412,A 0.000,B 0.000,C 90.000,E1 110.066} C_DIS
LIN {X 0.112,Y -574.275,Z 1159.410,A 0.000,B 0.000,C 90.000,E1 109.704} C_DIS
LIN {X -0.109,Y -568.255,Z 1159.407,A 0.000,B 0.000,C 90.000,E1 109.268} C_DIS
LIN {X -0.027,Y -560.355,Z 1159.404,A 0.000,B 0.000,C 90.000,E1 108.725} C_DIS
LIN {X -0.010,Y -555.662,Z 1159.402,A 0.000,B 0.000,C 90.000,E1 108.417} C_DIS
LIN {X 0.117,Y -551.453,Z 1159.400,A 0.000,B 0.000,C 90.000,E1 108.055} C_DIS
LIN {X -0.035,Y -550.249,Z 1159.399,A 0.000,B 0.000,C 90.000,E1 107.873} C_DIS
LIN {X -0.077,Y -550.244,Z 1159.399,A 0.000,B 0.000,C 90.000,E1 107.873} C_DIS
LIN {X -0.233,Y -549.962,Z 1159.398,A 0.000,B 0.000,C 90.000,E1 107.583} C_DIS
LIN {X -0.180,Y -550.398,Z 1159.393,A 0.000,B 0.000,C 90.000,E1 106.677} C_DIS
LIN {X 0.220,Y -551.723,Z 1159.383,A 0.000,B 0.000,C 90.000,E1 104.954} C_DIS
LIN {X 0.097,Y -553.331,Z 1159.372,A 0.000,B 0.000,C 90.000,E1 103.008} C_DIS
LIN {X 0.027,Y -555.498,Z 1159.360,A 0.000,B 0.000,C 90.000,E1 100.782} C_DIS
LIN {X 0.006,Y -556.533,Z 1159.354,A 0.000,B 0.000,C 90.000,E1 99.670} C_DIS
LIN {X 0.036,Y -557.829,Z 1159.346,A 0.000,B 0.000,C 90.000,E1 98.276} C_DIS
LIN {X 0.006,Y -559.005,Z 1159.338,A 0.000,B 0.000,C 90.000,E1 96.891} C_DIS
LIN {X 0.074,Y -560.238,Z 1159.329,A 0.000,B 0.000,C 90.000,E1 95.220} C_DIS
LIN {X 0.216,Y -561.625,Z 1159.318,A 0.000,B 0.000,C 90.000,E1 93.269} C_DIS
LIN {X -0.171,Y -563.139,Z 1159.308,A 0.000,B 0.000,C 90.000,E1 91.375} C_DIS
LIN {X 0.005,Y -564.576,Z 1159.297,A 0.000,B 0.000,C 90.000,E1 89.427} C_DIS
LIN {X 0.117,Y -565.591,Z 1159.288,A 0.000,B 0.000,C 90.000,E1 87.764} C_DIS
LIN {X 0.138,Y -566.426,Z 1159.280,A 0.000,B 0.000,C 90.000,E1 86.388} C_DIS
LIN {X -0.089,Y -567.544,Z 1159.269,A 0.000,B 0.000,C 90.000,E1 84.489} C_DIS
LIN {X -0.002,Y -568.424,Z 1159.262,A 0.000,B 0.000,C 90.000,E1 83.109} C_DIS
LIN {X -0.228,Y -569.365,Z 1159.253,A 0.000,B 0.000,C 90.000,E1 81.489} C_DIS
LIN {X 0.220,Y -570.111,Z 1159.244,A 0.000,B 0.000,C 90.000,E1 79.803} C_DIS
LIN {X 0.120,Y -570.933,Z 1159.234,A 0.000,B 0.000,C 90.000,E1 78.173} C_DIS
LIN {X 0.142,Y -571.696,Z 1159.225,A 0.000,B 0.000,C 90.000,E1 76.533} C_DIS
LIN {X -0.245,Y -572.499,Z 1159.216,A 0.000,B 0.000,C 90.000,E1 74.936} C_DIS
LIN {X 0.077,Y -573.744,Z 1159.204,A 0.000,B 0.000,C 90.000,E1 72.725} C_DIS
LIN {X -0.293,Y -574.296,Z 1159.200,A 0.000,B 0.000,C 90.000,E1 71.945} C_DIS
LIN {X 0.273,Y -576.059,Z 1159.186,A 0.000,B 0.000,C 90.000,E1 69.444} C_DIS
LIN {X -0.185,Y -577.694,Z 1159.175,A 0.000,B 0.000,C 90.000,E1 67.592} C_DIS
LIN {X 0.293,Y -579.335,Z 1159.166,A 0.000,B 0.000,C 90.000,E1 65.921} C_DIS
LIN {X -0.155,Y -581.020,Z 1159.156,A 0.000,B 0.000,C 90.000,E1 64.076} C_DIS
LIN {X -0.303,Y -582.328,Z 1159.148,A 0.000,B 0.000,C 90.000,E1 62.743} C_DIS
LIN {X -0.170,Y -583.569,Z 1159.141,A 0.000,B 0.000,C 90.000,E1 61.385} C_DIS
LIN {X 0.265,Y -584.715,Z 1159.134,A 0.000,B 0.000,C 90.000,E1 59.999} C_DIS
LIN {X 0.219,Y -585.744,Z 1159.126,A 0.000,B 0.000,C 90.000,E1 58.663} C_DIS
LIN {X 0.370,Y -586.801,Z 1159.117,A 0.000,B 0.000,C 90.000,E1 57.041} C_DIS
LIN {X -0.009,Y -587.563,Z 1159.111,A 0.000,B 0.000,C 90.000,E1 56.008} C_DIS
LIN {X 0.013,Y -588.519,Z 1159.102,A 0.000,B 0.000,C 90.000,E1 54.402} C_DIS
LIN {X -0.020,Y -589.778,Z 1159.090,A 0.000,B 0.000,C 90.000,E1 52.271} C_DIS
LIN {X 0.335,Y -590.347,Z 1159.084,A 0.000,B 0.000,C 90.000,E1 51.170} C_DIS
LIN {X 0.068,Y -590.977,Z 1159.077,A 0.000,B 0.000,C 90.000,E1 49.865} C_DIS
LIN {X 0.368,Y -591.258,Z 1159.071,A 0.000,B 0.000,C 90.000,E1 48.771} C_DIS
LIN {X -0.152,Y -591.481,Z 1159.065,A 0.000,B 0.000,C 90.000,E1 47.757} C_DIS
LIN {X -0.066,Y -591.546,Z 1159.058,A 0.000,B 0.000,C 90.000,E1 46.419} C_DIS
LIN {X 0.017,Y -591.379,Z 1159.051,A 0.000,B 0.000,C 90.000,E1 45.081} C_DIS
LIN {X -0.094,Y -591.041,Z 1159.045,A 0.000,B 0.000,C 90.000,E1 44.028} C_DIS
LIN {X 0.216,Y -590.427,Z 1159.039,A 0.000,B 0.000,C 90.000,E1 42.933} C_DIS
LIN {X -0.266,Y -590.145,Z 1159.036,A 0.000,B 0.000,C 90.000,E1 42.447} C_DIS
LIN {X 0.024,Y -589.220,Z 1159.030,A 0.000,B 0.000,C 90.000,E1 41.353} C_DIS
LIN {X 0.104,Y -587.825,Z 1159.022,A 0.000,B 0.000,C 90.000,E1 40.011} C_DIS
LIN {X 0.234,Y -586.868,Z 1159.018,A 0.000,B 0.000,C 90.000,E1 39.197} C_DIS
LIN {X -0.090,Y -585.067,Z 1159.010,A 0.000,B 0.000,C 90.000,E1 37.890} C_DIS
LIN {X 0.190,Y -583.384,Z 1159.005,A 0.000,B 0.000,C 90.000,E1 36.790} C_DIS
LIN {X -0.073,Y -580.634,Z 1158.997,A 0.000,B 0.000,C 90.000,E1 35.471} C_DIS
LIN {X -0.043,Y -578.597,Z 1158.993,A 0.000,B 0.000,C 90.000,E1 34.659} C_DIS
LIN {X -0.049,Y -577.156,Z 1158.990,A 0.000,B 0.000,C 90.000,E1 34.119} C_DIS
LIN {X 0.088,Y -574.601,Z 1158.985,A 0.000,B 0.000,C 90.000,E1 33.293} C_DIS
LIN {X 0.060,Y -572.763,Z 1158.982,A 0.000,B 0.000,C 90.000,E1 32.752} C_DIS
LIN {X -0.033,Y -568.592,Z 1158.976,A 0.000,B 0.000,C 90.000,E1 31.671} C_DIS
LIN {X 0.002,Y -564.883,Z 1158.971,A 0.000,B 0.000,C 90.000,E1 30.846} C_DIS
LIN {X 0.102,Y -562.246,Z 1158.968,A 0.000,B 0.000,C 90.000,E1 30.285} C_DIS
LIN {X -0.049,Y -557.184,Z 1158.963,A 0.000,B 0.000,C 90.000,E1 29.333} C_DIS
LIN {X 0.170,Y -553.278,Z 1158.959,A 0.000,B 0.000,C 90.000,E1 28.615} C_DIS
LIN {X 0.090,Y -549.002,Z 1158.955,A 0.000,B 0.000,C 90.000,E1 27.924} C_DIS
LIN {X -0.128,Y -545.345,Z 1158.952,A 0.000,B 0.000,C 90.000,E1 27.385} C_DIS
LIN {X 0.106,Y -541.411,Z 1158.949,A 0.000,B 0.000,C 90.000,E1 26.796} C_DIS
LIN {X -0.067,Y -536.135,Z 1158.945,A 0.000,B 0.000,C 90.000,E1 26.104} C_DIS
LIN {X -0.281,Y -530.506,Z 1158.941,A 0.000,B 0.000,C 90.000,E1 25.412} C_DIS
LIN {X 0.160,Y -524.472,Z 1158.937,A 0.000,B 0.000,C 90.000,E1 24.643} C_DIS
LIN {X -0.212,Y -516.854,Z 1158.932,A 0.000,B 0.000,C 90.000,E1 23.823} C_DIS
LIN {X 0.051,Y -510.071,Z 1158.928,A 0.000,B 0.000,C 90.000,E1 23.078} C_DIS
LIN {X -0.108,Y -501.850,Z 1158.924,A 0.000,B 0.000,C 90.000,E1 22.259} C_DIS
LIN {X 0.215,Y -493.292,Z 1158.919,A 0.000,B 0.000,C 90.000,E1 21.408} C_DIS
LIN {X -0.158,Y -487.547,Z 1158.916,A 0.000,B 0.000,C 90.000,E1 20.918} C_DIS
LIN {X -0.140,Y -477.341,Z 1158.911,A 0.000,B 0.000,C 90.000,E1 19.993} C_DIS
LIN {X 0.187,Y -465.726,Z 1158.905,A 0.000,B 0.000,C 90.000,E1 18.906} C_DIS
LIN {X 0.034,Y -449.398,Z 1158.897,A 0.000,B 0.000,C 90.000,E1 17.457} C_DIS
LIN {X -0.183,Y -431.968,Z 1158.888,A 0.000,B 0.000,C 90.000,E1 15.788} C_DIS
LIN {X -0.143,Y -419.297,Z 1158.880,A 0.000,B 0.000,C 90.000,E1 14.411} C_DIS
LIN {X 0.166,Y -408.346,Z 1158.873,A 0.000,B 0.000,C 90.000,E1 13.063} C_DIS
LIN {X -0.098,Y -400.700,Z 1158.867,A 0.000,B 0.000,C 90.000,E1 12.063} C_DIS
LIN {X -0.072,Y -397.244,Z 1158.864,A 0.000,B 0.000,C 90.000,E1 11.535} C_DIS
LIN {X -0.069,Y -394.328,Z 1158.861,A 0.000,B 0.000,C 90.000,E1 11.007} C_DIS
LIN {X -0.076,Y -392.810,Z 1158.859,A 0.000,B 0.000,C 90.000,E1 10.602} C_DIS
LIN {X -0.185,Y -392.541,Z 1158.857,A 0.000,B 0.000,C 90.000,E1 10.197} C_DIS
LIN {X -0.050,Y -393.541,Z 1158.853,A 0.000,B 0.000,C 90.000,E1 9.557} C_DIS
LIN {X -0.118,Y -396.058,Z 1158.848,A 0.000,B 0.000,C 90.000,E1 8.681} C_DIS
LIN {X 0.147,Y -400.327,Z 1158.841,A 0.000,B 0.000,C 90.000,E1 7.409} C_DIS
LIN {X 0.080,Y -401.637,Z 1158.839,A 0.000,B 0.000,C 90.000,E1 7.068} C_DIS
LIN {X 0.115,Y -403.670,Z 1158.837,A 0.000,B 0.000,C 90.000,E1 6.663} C_DIS
LIN {X -0.196,Y -406.597,Z 1158.834,A 0.000,B 0.000,C 90.000,E1 6.201} C_DIS
LIN {X -0.175,Y -407.917,Z 1158.833,A 0.000,B 0.000,C 90.000,E1 6.024} C_DIS
LIN {X -0.149,Y -411.100,Z 1158.832,A 0.000,B 0.000,C 90.000,E1 5.682} C_DIS
LIN {X 0.002,Y -415.058,Z 1158.830,A 0.000,B 0.000,C 90.000,E1 5.334} C_DIS
LIN {X -0.083,Y -434.515,Z 1158.822,A 0.000,B 0.000,C 90.000,E1 3.898} C_DIS
LIN {X -0.094,Y -457.128,Z 1158.813,A 0.000,B 0.000,C 90.000,E1 2.293} C_DIS
LIN {X -0.201,Y -471.651,Z 1158.807,A 0.000,B 0.000,C 90.000,E1 1.318} C_DIS
LIN {X -0.068,Y -477.954,Z 1158.805,A 0.000,B 0.000,C 90.000,E1 0.859} C_DIS
LIN {X 0.000,Y -489.349,Z 1158.800,A 0.000,B 0.000,C 90.000,E1 360.000} C_DIS
LIN {X 0.009,Y -496.489,Z 1158.797,A 0.000,B 0.000,C 90.000,E1 359.427} C_DIS
LIN {X -0.007,Y -503.730,Z 1158.793,A 0.000,B 0.000,C 90.000,E1 358.797} C_DIS
LIN {X -0.208,Y -510.533,Z 1158.790,A 0.000,B 0.000,C 90.000,E1 358.165} C_DIS
LIN {X -0.216,Y -517.031,Z 1158.786,A 0.000,B 0.000,C 90.000,E1 357.478} C_DIS
LIN {X -0.270,Y -522.203,Z 1158.783,A 0.000,B 0.000,C 90.000,E1 356.906} C_DIS
LIN {X -0.001,Y -528.083,Z 1158.779,A 0.000,B 0.000,C 90.000,E1 356.159} C_DIS
LIN {X -0.256,Y -533.417,Z 1158.775,A 0.000,B 0.000,C 90.000,E1 355.469} C_DIS
LIN {X 0.024,Y -538.104,Z 1158.771,A 0.000,B 0.000,C 90.000,E1 354.723} C_DIS
LIN {X -0.193,Y -542.425,Z 1158.767,A 0.000,B 0.000,C 90.000,E1 354.033} C_DIS
LIN {X -0.050,Y -545.563,Z 1158.764,A 0.000,B 0.000,C 90.000,E1 353.451} C_DIS
LIN {X -0.201,Y -549.166,Z 1158.760,A 0.000,B 0.000,C 90.000,E1 352.761} C_DIS
LIN {X 0.038,Y -553.016,Z 1158.755,A 0.000,B 0.000,C 90.000,E1 351.894} C_DIS
LIN {X 0.022,Y -555.879,Z 1158.751,A 0.000,B 0.000,C 90.000,E1 351.197} C_DIS
LIN {X -0.224,Y -558.958,Z 1158.746,A 0.000,B 0.000,C 90.000,E1 350.387} C_DIS
LIN {X 0.210,Y -561.731,Z 1158.742,A 0.000,B 0.000,C 90.000,E1 349.511} C_DIS
LIN {X 0.017,Y -564.300,Z 1158.737,A 0.000,B 0.000,C 90.000,E1 348.701} C_DIS
LIN {X 0.127,Y -567.390,Z 1158.731,A 0.000,B 0.000,C 90.000,E1 347.589} C_DIS
LIN {X 0.228,Y -569.574,Z 1158.727,A 0.000,B 0.000,C 90.000,E1 346.756} C_DIS
LIN {X -0.142,Y -572.361,Z 1158.721,A 0.000,B 0.000,C 90.000,E1 345.700} C_DIS
LIN {X 0.219,Y -574.992,Z 1158.714,A 0.000,B 0.000,C 90.000,E1 344.574} C_DIS
LIN {X 0.061,Y -577.475,Z 1158.708,A 0.000,B 0.000,C 90.000,E1 343.504} C_DIS
LIN {X 0.104,Y -579.857,Z 1158.702,A 0.000,B 0.000,C 90.000,E1 342.417} C_DIS
LIN {X 0.187,Y -582.184,Z 1158.696,A 0.000,B 0.000,C 90.000,E1 341.329} C_DIS
LIN {X -0.042,Y -584.717,Z 1158.689,A 0.000,B 0.000,C 90.000,E1 340.007} C_DIS
LIN {X 0.173,Y -586.899,Z 1158.682,A 0.000,B 0.000,C 90.000,E1 338.646} C_DIS
LIN {X 0.128,Y -588.031,Z 1158.677,A 0.000,B 0.000,C 90.000,E1 337.847} C_DIS
LIN {X -0.025,Y -589.115,Z 1158.671,A 0.000,B 0.000,C 90.000,E1 336.794} C_DIS
LIN {X 0.181,Y -589.692,Z 1158.667,A 0.000,B 0.000,C 90.000,E1 335.973} C_DIS
LIN {X 0.150,Y -590.005,Z 1158.662,A 0.000,B 0.000,C 90.000,E1 335.177} C_DIS
LIN {X -0.171,Y -590.020,Z 1158.658,A 0.000,B 0.000,C 90.000,E1 334.409} C_DIS
LIN {X 0.039,Y -589.709,Z 1158.653,A 0.000,B 0.000,C 90.000,E1 333.589} C_DIS
LIN {X -0.014,Y -589.046,Z 1158.649,A 0.000,B 0.000,C 90.000,E1 332.794} C_DIS
LIN {X -0.229,Y -588.402,Z 1158.646,A 0.000,B 0.000,C 90.000,E1 332.281} C_DIS
LIN {X 0.068,Y -587.586,Z 1158.643,A 0.000,B 0.000,C 90.000,E1 331.719} C_DIS
LIN {X -0.117,Y -585.399,Z 1158.637,A 0.000,B 0.000,C 90.000,E1 330.667} C_DIS
LIN {X -0.202,Y -583.267,Z 1158.633,A 0.000,B 0.000,C 90.000,E1 329.871} C_DIS
LIN {X -0.307,Y -580.657,Z 1158.628,A 0.000,B 0.000,C 90.000,E1 329.076} C_DIS
LIN {X -0.137,Y -577.482,Z 1158.624,A 0.000,B 0.000,C 90.000,E1 328.250} C_DIS
LIN {X -0.225,Y -574.152,Z 1158.620,A 0.000,B 0.000,C 90.000,E1 327.582} C_DIS
LIN {X -0.345,Y -570.154,Z 1158.616,A 0.000,B 0.000,C 90.000,E1 326.914} C_DIS
LIN {X -0.191,Y -565.650,Z 1158.612,A 0.000,B 0.000,C 90.000,E1 326.215} C_DIS
LIN {X -0.285,Y -561.788,Z 1158.609,A 0.000,B 0.000,C 90.000,E1 325.674} C_DIS
LIN {X -0.002,Y -555.246,Z 1158.605,A 0.000,B 0.000,C 90.000,E1 324.815} C_DIS
LIN {X -0.046,Y -551.726,Z 1158.602,A 0.000,B 0.000,C 90.000,E1 324.402} C_DIS
LIN {X 0.128,Y -544.321,Z 1158.598,A 0.000,B 0.000,C 90.000,E1 323.543} C_DIS
LIN {X 0.154,Y -537.882,Z 1158.594,A 0.000,B 0.000,C 90.000,E1 322.844} C_DIS
LIN {X -0.066,Y -530.505,Z 1158.589,A 0.000,B 0.000,C 90.000,E1 322.065} C_DIS
LIN {X 0.215,Y -527.090,Z 1158.587,A 0.000,B 0.000,C 90.000,E1 321.618} C_DIS
LIN {X 0.189,Y -524.890,Z 1158.585,A 0.000,B 0.000,C 90.000,E1 321.331} C_DIS
LIN {X -0.107,Y -522.349,Z 1158.583,A 0.000,B 0.000,C 90.000,E1 320.928} C_DIS
LIN {X -0.200,Y -521.191,Z 1158.581,A 0.000,B 0.000,C 90.000,E1 320.642} C_DIS
LIN {X -0.248,Y -520.188,Z 1158.580,A 0.000,B 0.000,C 90.000,E1 320.356} C_DIS
LIN {X 0.112,Y -519.120,Z 1158.576,A 0.000,B 0.000,C 90.000,E1 319.703} C_DIS
LIN {X 0.088,Y -518.895,Z 1158.571,A 0.000,B 0.000,C 90.000,E1 318.728} C_DIS
LIN {X -0.275,Y -519.905,Z 1158.556,A 0.000,B 0.000,C 90.000,E1 316.134} C_DIS
LIN {X -0.008,Y -520.779,Z 1158.546,A 0.000,B 0.000,C 90.000,E1 314.352} C_DIS
LIN {X -0.023,Y -521.473,Z 1158.538,A 0.000,B 0.000,C 90.000,E1 312.894} C_DIS
LIN {X -0.059,Y -522.414,Z 1158.529,A 0.000,B 0.000,C 90.000,E1 311.148} C_DIS
LIN {X -0.070,Y -523.357,Z 1158.519,A 0.000,B 0.000,C 90.000,E1 309.402} C_DIS
LIN {X -0.033,Y -524.560,Z 1158.508,A 0.000,B 0.000,C 90.000,E1 307.363} C_DIS
LIN {X -0.179,Y -525.308,Z 1158.501,A 0.000,B 0.000,C 90.000,E1 306.217} C_DIS
LIN {X 0.041,Y -526.295,Z 1158.491,A 0.000,B 0.000,C 90.000,E1 304.452} C_DIS
LIN {X 0.069,Y -527.777,Z 1158.479,A 0.000,B 0.000,C 90.000,E1 302.133} C_DIS
LIN {X 0.240,Y -528.686,Z 1158.471,A 0.000,B 0.000,C 90.000,E1 300.669} C_DIS
LIN {X 0.010,Y -529.423,Z 1158.464,A 0.000,B 0.000,C 90.000,E1 299.539} C_DIS
LIN {X -0.171,Y -529.848,Z 1158.459,A 0.000,B 0.000,C 90.000,E1 298.693} C_DIS
LIN {X -0.223,Y -530.391,Z 1158.451,A 0.000,B 0.000,C 90.000,E1 297.257} C_DIS
LIN {X -0.035,Y -530.686,Z 1158.443,A 0.000,B 0.000,C 90.000,E1 295.796} C_DIS
LIN {X 0.160,Y -530.776,Z 1158.435,A 0.000,B 0.000,C 90.000,E1 294.335} C_DIS
LIN {X 0.025,Y -530.699,Z 1158.424,A 0.000,B 0.000,C 90.000,E1 292.333} C_DIS
LIN {X -0.207,Y -530.649,Z 1158.416,A 0.000,B 0.000,C 90.000,E1 290.918} C_DIS
LIN {X 0.241,Y -530.229,Z 1158.406,A 0.000,B 0.000,C 90.000,E1 289.141} C_DIS
LIN {X 0.134,Y -529.848,Z 1158.400,A 0.000,B 0.000,C 90.000,E1 288.000} C_DIS
LIN {X 0.221,Y -529.139,Z 1158.391,A 0.000,B 0.000,C 90.000,E1 286.260} C_DIS
LIN {X -0.046,Y -528.605,Z 1158.384,A 0.000,B 0.000,C 90.000,E1 285.134} C_DIS
LIN {X -0.165,Y -527.873,Z 1158.376,A 0.000,B 0.000,C 90.000,E1 283.703} C_DIS
LIN {X -0.061,Y -527.199,Z 1158.370,A 0.000,B 0.000,C 90.000,E1 282.535} C_DIS
LIN {X 0.089,Y -526.071,Z 1158.360,A 0.000,B 0.000,C 90.000,E1 280.782} C_DIS
LIN {X 0.205,Y -524.917,Z 1158.350,A 0.000,B 0.000,C 90.000,E1 279.029} C_DIS
LIN {X 0.177,Y -524.218,Z 1158.344,A 0.000,B 0.000,C 90.000,E1 277.871} C_DIS
LIN {X 0.075,Y -523.340,Z 1158.336,A 0.000,B 0.000,C 90.000,E1 276.429} C_DIS
LIN {X -0.100,Y -522.486,Z 1158.326,A 0.000,B 0.000,C 90.000,E1 274.702} C_DIS
LIN {X 0.207,Y -521.842,Z 1158.318,A 0.000,B 0.000,C 90.000,E1 273.212} C_DIS
LIN {X -0.043,Y -521.159,Z 1158.308,A 0.000,B 0.000,C 90.000,E1 271.489} C_DIS
LIN {X 0.231,Y -520.532,Z 1158.300,A 0.000,B 0.000,C 90.000,E1 270.000} C_DIS
LIN {X -0.027,Y -519.911,Z 1158.292,A 0.000,B 0.000,C 90.000,E1 268.568} C_DIS
LIN {X 0.200,Y -519.101,Z 1158.282,A 0.000,B 0.000,C 90.000,E1 266.788} C_DIS
LIN {X -0.009,Y -518.387,Z 1158.276,A 0.000,B 0.000,C 90.000,E1 265.641} C_DIS
LIN {X -0.264,Y -517.313,Z 1158.268,A 0.000,B 0.000,C 90.000,E1 264.204} C_DIS
LIN {X 0.005,Y -515.593,Z 1158.258,A 0.000,B 0.000,C 90.000,E1 262.413} C_DIS
LIN {X -0.278,Y -513.859,Z 1158.248,A 0.000,B 0.000,C 90.000,E1 260.679} C_DIS
LIN {X 0.075,Y -512.140,Z 1158.238,A 0.000,B 0.000,C 90.000,E1 258.870} C_DIS
LIN {X -0.150,Y -510.256,Z 1158.227,A 0.000,B 0.000,C 90.000,E1 256.825} C_DIS
LIN {X -0.189,Y -509.235,Z 1158.220,A 0.000,B 0.000,C 90.000,E1 255.644} C_DIS
LIN {X -0.070,Y -507.729,Z 1158.210,A 0.000,B 0.000,C 90.000,E1 253.850} C_DIS
LIN {X 0.022,Y -506.062,Z 1158.200,A 0.000,B 0.000,C 90.000,E1 252.054} C_DIS
LIN {X 0.225,Y -504.362,Z 1158.190,A 0.000,B 0.000,C 90.000,E1 250.242} C_DIS
LIN {X 0.083,Y -502.587,Z 1158.180,A 0.000,B 0.000,C 90.000,E1 248.465} C_DIS
LIN {X -0.141,Y -501.766,Z 1158.175,A 0.000,B 0.000,C 90.000,E1 247.592} C_DIS
LIN {X 0.232,Y -500.018,Z 1158.167,A 0.000,B 0.000,C 90.000,E1 246.049} C_DIS
LIN {X -0.142,Y -498.147,Z 1158.159,A 0.000,B 0.000,C 90.000,E1 244.588} C_DIS
LIN {X 0.165,Y -495.700,Z 1158.149,A 0.000,B 0.000,C 90.000,E1 242.743} C_DIS
LIN {X 0.196,Y -493.115,Z 1158.139,A 0.000,B 0.000,C 90.000,E1 240.923} C_DIS
LIN {X -0.106,Y -491.307,Z 1158.132,A 0.000,B 0.000,C 90.000,E1 239.744} C_DIS
LIN {X 0.063,Y -489.057,Z 1158.123,A 0.000,B 0.000,C 90.000,E1 238.201} C_DIS
LIN {X -0.164,Y -485.786,Z 1158.112,A 0.000,B 0.000,C 90.000,E1 236.087} C_DIS
LIN {X 0.069,Y -482.550,Z 1158.100,A 0.000,B 0.000,C 90.000,E1 233.909} C_DIS
LIN {X 0.011,Y -480.665,Z 1158.093,A 0.000,B 0.000,C 90.000,E1 232.683} C_DIS
LIN {X 0.105,Y -476.784,Z 1158.079,A 0.000,B 0.000,C 90.000,E1 230.194} C_DIS
LIN {X 0.135,Y -473.881,Z 1158.069,A 0.000,B 0.000,C 90.000,E1 228.324} C_DIS
LIN {X 0.052,Y -470.798,Z 1158.058,A 0.000,B 0.000,C 90.000,E1 226.458} C_DIS
LIN {X -0.134,Y -464.392,Z 1158.032,A 0.000,B 0.000,C 90.000,E1 221.757} C_DIS
LIN {X 0.068,Y -462.305,Z 1158.018,A 0.000,B 0.000,C 90.000,E1 219.197} C_DIS
LIN {X -0.125,Y -460.886,Z 1158.005,A 0.000,B 0.000,C 90.000,E1 216.996} C_DIS
LIN {X 0.116,Y -459.485,Z 1157.967,A 0.000,B 0.000,C 90.000,E1 209.951} C_DIS
LIN {X 0.218,Y -460.376,Z 1157.956,A 0.000,B 0.000,C 90.000,E1 208.025} C_DIS
LIN {X -0.150,Y -462.857,Z 1157.940,A 0.000,B 0.000,C 90.000,E1 205.207} C_DIS
LIN {X 0.223,Y -465.401,Z 1157.929,A 0.000,B 0.000,C 90.000,E1 203.259} C_DIS
LIN {X 0.067,Y -471.908,Z 1157.910,A 0.000,B 0.000,C 90.000,E1 199.812} C_DIS
LIN {X -0.232,Y -479.146,Z 1157.895,A 0.000,B 0.000,C 90.000,E1 197.040} C_DIS
LIN {X -0.087,Y -488.834,Z 1157.877,A 0.000,B 0.000,C 90.000,E1 193.939} C_DIS
LIN {X -0.161,Y -494.964,Z 1157.867,A 0.000,B 0.000,C 90.000,E1 192.119} C_DIS
LIN {X 0.225,Y -502.427,Z 1157.856,A 0.000,B 0.000,C 90.000,E1 189.962} C_DIS
LIN {X 0.113,Y -511.189,Z 1157.842,A 0.000,B 0.000,C 90.000,E1 187.587} C_DIS
LIN {X -0.193,Y -516.722,Z 1157.834,A 0.000,B 0.000,C 90.000,E1 186.144} C_DIS
LIN {X 0.110,Y -522.114,Z 1157.826,A 0.000,B 0.000,C 90.000,E1 184.645} C_DIS
LIN {X -0.090,Y -527.498,Z 1157.818,A 0.000,B 0.000,C 90.000,E1 183.212} C_DIS
LIN {X -0.168,Y -532.861,Z 1157.810,A 0.000,B 0.000,C 90.000,E1 181.776} C_DIS
LIN {X -0.192,Y -537.156,Z 1157.803,A 0.000,B 0.000,C 90.000,E1 180.630} C_DIS
LIN {X -0.105,Y -543.568,Z 1157.794,A 0.000,B 0.000,C 90.000,E1 178.912} C_DIS
LIN {X 0.180,Y -551.082,Z 1157.783,A 0.000,B 0.000,C 90.000,E1 176.906} C_DIS
LIN {X 0.055,Y -557.467,Z 1157.774,A 0.000,B 0.000,C 90.000,E1 175.241} C_DIS
LIN {X 0.032,Y -562.745,Z 1157.766,A 0.000,B 0.000,C 90.000,E1 173.856} C_DIS
LIN {X 0.209,Y -569.085,Z 1157.757,A 0.000,B 0.000,C 90.000,E1 172.186} C_DIS
LIN {X 0.222,Y -576.383,Z 1157.746,A 0.000,B 0.000,C 90.000,E1 170.274} C_DIS
LIN {X -0.293,Y -582.529,Z 1157.737,A 0.000,B 0.000,C 90.000,E1 168.701} C_DIS
LIN {X 0.080,Y -586.525,Z 1157.731,A 0.000,B 0.000,C 90.000,E1 167.589} C_DIS
LIN {X 0.075,Y -590.401,Z 1157.725,A 0.000,B 0.000,C 90.000,E1 166.520} C_DIS
LIN {X -0.011,Y -594.155,Z 1157.719,A 0.000,B 0.000,C 90.000,E1 165.463} C_DIS
LIN {X -0.194,Y -598.719,Z 1157.712,A 0.000,B 0.000,C 90.000,E1 164.157} C_DIS
LIN {X -0.023,Y -602.233,Z 1157.706,A 0.000,B 0.000,C 90.000,E1 163.087} C_DIS
LIN {X 0.101,Y -606.440,Z 1157.699,A 0.000,B 0.000,C 90.000,E1 161.764} C_DIS
LIN {X -0.016,Y -609.612,Z 1157.693,A 0.000,B 0.000,C 90.000,E1 160.732} C_DIS
LIN {X -0.138,Y -613.465,Z 1157.686,A 0.000,B 0.000,C 90.000,E1 159.444} C_DIS
LIN {X -0.163,Y -616.422,Z 1157.680,A 0.000,B 0.000,C 90.000,E1 158.411} C_DIS
LIN {X 0.047,Y -620.670,Z 1157.671,A 0.000,B 0.000,C 90.000,E1 156.847} C_DIS
LIN {X 0.349,Y -624.069,Z 1157.664,A 0.000,B 0.000,C 90.000,E1 155.537} C_DIS
LIN {X 0.149,Y -628.060,Z 1157.656,A 0.000,B 0.000,C 90.000,E1 154.024} C_DIS
LIN {X -0.230,Y -632.461,Z 1157.646,A 0.000,B 0.000,C 90.000,E1 152.281} C_DIS
LIN {X -0.047,Y -635.412,Z 1157.639,A 0.000,B 0.000,C 90.000,E1 151.001} C_DIS
LIN {X -0.115,Y -637.695,Z 1157.633,A 0.000,B 0.000,C 90.000,E1 149.999} C_DIS
LIN {X -0.096,Y -640.375,Z 1157.626,A 0.000,B 0.000,C 90.000,E1 148.742} C_DIS
LIN {X 0.300,Y -642.846,Z 1157.619,A 0.000,B 0.000,C 90.000,E1 147.454} C_DIS
LIN {X -0.281,Y -645.628,Z 1157.611,A 0.000,B 0.000,C 90.000,E1 146.008} C_DIS
LIN {X -0.340,Y -647.816,Z 1157.604,A 0.000,B 0.000,C 90.000,E1 144.769} C_DIS
LIN {X 0.007,Y -649.948,Z 1157.597,A 0.000,B 0.000,C 90.000,E1 143.497} C_DIS
LIN {X -0.222,Y -653.241,Z 1157.586,A 0.000,B 0.000,C 90.000,E1 141.537} C_DIS
LIN {X 0.057,Y -655.938,Z 1157.578,A 0.000,B 0.000,C 90.000,E1 140.033} C_DIS
LIN {X -0.037,Y -658.888,Z 1157.570,A 0.000,B 0.000,C 90.000,E1 138.566} C_DIS
LIN {X 0.343,Y -660.931,Z 1157.564,A 0.000,B 0.000,C 90.000,E1 137.553} C_DIS
LIN {X -0.211,Y -663.879,Z 1157.556,A 0.000,B 0.000,C 90.000,E1 136.134} C_DIS
LIN {X -0.235,Y -669.104,Z 1157.543,A 0.000,B 0.000,C 90.000,E1 133.704} C_DIS
LIN {X -0.109,Y -673.613,Z 1157.532,A 0.000,B 0.000,C 90.000,E1 131.757} C_DIS
LIN {X 0.225,Y -678.830,Z 1157.520,A 0.000,B 0.000,C 90.000,E1 129.564} C_DIS
LIN {X 0.032,Y -681.878,Z 1157.513,A 0.000,B 0.000,C 90.000,E1 128.382} C_DIS
LIN {X 0.425,Y -684.857,Z 1157.507,A 0.000,B 0.000,C 90.000,E1 127.156} C_DIS
LIN {X 0.091,Y -688.443,Z 1157.499,A 0.000,B 0.000,C 90.000,E1 125.758} C_DIS
LIN {X 0.225,Y -691.906,Z 1157.491,A 0.000,B 0.000,C 90.000,E1 124.326} C_DIS
LIN {X 0.336,Y -694.136,Z 1157.486,A 0.000,B 0.000,C 90.000,E1 123.372} C_DIS
LIN {X -0.106,Y -696.302,Z 1157.480,A 0.000,B 0.000,C 90.000,E1 122.467} C_DIS
LIN {X -0.309,Y -698.253,Z 1157.475,A 0.000,B 0.000,C 90.000,E1 121.544} C_DIS
LIN {X 0.143,Y -700.438,Z 1157.469,A 0.000,B 0.000,C 90.000,E1 120.335} C_DIS
LIN {X -0.059,Y -702.944,Z 1157.461,A 0.000,B 0.000,C 90.000,E1 118.949} C_DIS
LIN {X -0.174,Y -704.555,Z 1157.456,A 0.000,B 0.000,C 90.000,E1 118.025} C_DIS
LIN {X 0.059,Y -705.504,Z 1157.452,A 0.000,B 0.000,C 90.000,E1 117.308} C_DIS
LIN {X -0.311,Y -705.987,Z 1157.449,A 0.000,B 0.000,C 90.000,E1 116.873} C_DIS
LIN {X 0.212,Y -706.577,Z 1157.443,A 0.000,B 0.000,C 90.000,E1 115.668} C_DIS
LIN {X 0.157,Y -706.633,Z 1157.439,A 0.000,B 0.000,C 90.000,E1 114.975} C_DIS
LIN {X 0.102,Y -706.376,Z 1157.436,A 0.000,B 0.000,C 90.000,E1 114.515} C_DIS
LIN {X -0.249,Y -705.478,Z 1157.434,A 0.000,B 0.000,C 90.000,E1 114.079} C_DIS
LIN {X 0.040,Y -704.823,Z 1157.432,A 0.000,B 0.000,C 90.000,E1 113.823} C_DIS
LIN {X -0.317,Y -702.752,Z 1157.430,A 0.000,B 0.000,C 90.000,E1 113.387} C_DIS
LIN {X -0.178,Y -702.074,Z 1157.429,A 0.000,B 0.000,C 90.000,E1 113.259} C_DIS
LIN {X 0.091,Y -697.728,Z 1157.427,A 0.000,B 0.000,C 90.000,E1 112.770} C_DIS
LIN {X 0.221,Y -696.471,Z 1157.426,A 0.000,B 0.000,C 90.000,E1 112.642} C_DIS
LIN {X 0.393,Y -694.593,Z 1157.425,A 0.000,B 0.000,C 90.000,E1 112.514} C_DIS
LIN {X -0.265,Y -685.952,Z 1157.424,A 0.000,B 0.000,C 90.000,E1 112.280} C_DIS
LIN {X 0.294,Y -684.607,Z 1157.424,A 0.000,B 0.000,C 90.000,E1 112.206} C_DIS
LIN {X 0.240,Y -676.706,Z 1157.423,A 0.000,B 0.000,C 90.000,E1 112.153} C_DIS
LIN {X 0.176,Y -604.054,Z 1157.423,A 0.000,B 0.000,C 90.000,E1 112.153} C_DIS
LIN {X -0.025,Y -600.965,Z 1157.422,A 0.000,B 0.000,C 90.000,E1 111.972} C_DIS
LIN {X 0.160,Y -595.494,Z 1157.420,A 0.000,B 0.000,C 90.000,E1 111.535} C_DIS
LIN {X 0.203,Y -577.129,Z 1157.411,A 0.000,B 0.000,C 90.000,E1 109.939} C_DIS
LIN {X 0.144,Y -574.318,Z 1157.410,A 0.000,B 0.000,C 90.000,E1 109.704} C_DIS
LIN {X -0.083,Y -568.294,Z 1157.407,A 0.000,B 0.000,C 90.000,E1 109.268} C_DIS
LIN {X -0.005,Y -560.327,Z 1157.404,A 0.000,B 0.000,C 90.000,E1 108.725} C_DIS
LIN {X 0.127,Y -555.786,Z 1157.402,A 0.000,B 0.000,C 90.000,E1 108.417} C_DIS
LIN {X 0.260,Y -551.493,Z 1157.401,A 0.000,B 0.000,C 90.000,E1 108.055} C_DIS
LIN {X -0.018,Y -550.224,Z 1157.399,A 0.000,B 0.000,C 90.000,E1 107.873} C_DIS
LIN {X -0.060,Y -550.215,Z 1157.399,A 0.000,B 0.000,C 90.000,E1 107.873} C_DIS
LIN {X -0.090,Y -549.944,Z 1157.398,A 0.000,B 0.000,C 90.000,E1 107.583} C_DIS
LIN {X -0.038,Y -550.357,Z 1157.393,A 0.000,B 0.000,C 90.000,E1 106.677} C_DIS
LIN {X -0.171,Y -551.652,Z 1157.383,A 0.000,B 0.000,C 90.000,E1 105.009} C_DIS
LIN {X -0.179,Y -553.539,Z 1157.371,A 0.000,B 0.000,C 90.000,E1 102.771} C_DIS
LIN {X -0.249,Y -555.697,Z 1157.359,A 0.000,B 0.000,C 90.000,E1 100.546} C_DIS
LIN {X -0.095,Y -557.225,Z 1157.349,A 0.000,B 0.000,C 90.000,E1 98.859} C_DIS
LIN {X -0.055,Y -558.455,Z 1157.342,A 0.000,B 0.000,C 90.000,E1 97.466} C_DIS
LIN {X -0.209,Y -559.289,Z 1157.335,A 0.000,B 0.000,C 90.000,E1 96.372} C_DIS
LIN {X -0.137,Y -560.561,Z 1157.326,A 0.000,B 0.000,C 90.000,E1 94.702} C_DIS
LIN {X 0.007,Y -561.952,Z 1157.315,A 0.000,B 0.000,C 90.000,E1 92.751} C_DIS
LIN {X -0.041,Y -563.068,Z 1157.308,A 0.000,B 0.000,C 90.000,E1 91.375} C_DIS
LIN {X 0.027,Y -564.272,Z 1157.298,A 0.000,B 0.000,C 90.000,E1 89.714} C_DIS
LIN {X -0.103,Y -565.002,Z 1157.292,A 0.000,B 0.000,C 90.000,E1 88.625} C_DIS
LIN {X 0.013,Y -565.993,Z 1157.283,A 0.000,B 0.000,C 90.000,E1 86.963} C_DIS
LIN {X 0.177,Y -566.946,Z 1157.274,A 0.000,B 0.000,C 90.000,E1 85.298} C_DIS
LIN {X -0.152,Y -567.986,Z 1157.265,A 0.000,B 0.000,C 90.000,E1 83.685} C_DIS
LIN {X 0.181,Y -568.906,Z 1157.256,A 0.000,B 0.000,C 90.000,E1 82.008} C_DIS
LIN {X 0.073,Y -569.332,Z 1157.251,A 0.000,B 0.000,C 90.000,E1 81.197} C_DIS
LIN {X -0.224,Y -569.971,Z 1157.244,A 0.000,B 0.000,C 90.000,E1 79.859} C_DIS
LIN {X 0.235,Y -570.787,Z 1157.234,A 0.000,B 0.000,C 90.000,E1 78.173} C_DIS
LIN {X 0.023,Y -571.675,Z 1157.224,A 0.000,B 0.000,C 90.000,E1 76.284} C_DIS
LIN {X 0.202,Y -572.507,Z 1157.215,A 0.000,B 0.000,C 90.000,E1 74.629} C_DIS
LIN {X 0.174,Y -573.979,Z 1157.201,A 0.000,B 0.000,C 90.000,E1 72.181} C_DIS
LIN {X -0.001,Y -575.714,Z 1157.188,A 0.000,B 0.000,C 90.000,E1 69.752} C_DIS
LIN {X -0.089,Y -577.582,Z 1157.176,A 0.000,B 0.000,C 90.000,E1 67.592} C_DIS
LIN {X 0.003,Y -578.917,Z 1157.168,A 0.000,B 0.000,C 90.000,E1 66.230} C_DIS
LIN {X 0.348,Y -580.147,Z 1157.161,A 0.000,B 0.000,C 90.000,E1 64.845} C_DIS
LIN {X 0.188,Y -581.384,Z 1157.153,A 0.000,B 0.000,C 90.000,E1 63.512} C_DIS
LIN {X -0.347,Y -582.396,Z 1157.147,A 0.000,B 0.000,C 90.000,E1 62.487} C_DIS
LIN {X -0.084,Y -583.409,Z 1157.141,A 0.000,B 0.000,C 90.000,E1 61.385} C_DIS
LIN {X -0.157,Y -584.544,Z 1157.134,A 0.000,B 0.000,C 90.000,E1 60.049} C_DIS
LIN {X 0.300,Y -585.576,Z 1157.126,A 0.000,B 0.000,C 90.000,E1 58.663} C_DIS
LIN {X -0.044,Y -586.622,Z 1157.117,A 0.000,B 0.000,C 90.000,E1 57.089} C_DIS
LIN {X -0.072,Y -587.499,Z 1157.110,A 0.000,B 0.000,C 90.000,E1 55.754} C_DIS
LIN {X 0.085,Y -588.327,Z 1157.102,A 0.000,B 0.000,C 90.000,E1 54.402} C_DIS
LIN {X -0.155,Y -589.400,Z 1157.092,A 0.000,B 0.000,C 90.000,E1 52.557} C_DIS
LIN {X 0.194,Y -590.004,Z 1157.086,A 0.000,B 0.000,C 90.000,E1 51.457} C_DIS
LIN {X -0.074,Y -590.644,Z 1157.079,A 0.000,B 0.000,C 90.000,E1 50.150} C_DIS
LIN {X -0.166,Y -590.965,Z 1157.073,A 0.000,B 0.000,C 90.000,E1 49.094} C_DIS
LIN {X -0.099,Y -591.232,Z 1157.065,A 0.000,B 0.000,C 90.000,E1 47.757} C_DIS
LIN {X -0.017,Y -591.263,Z 1157.058,A 0.000,B 0.000,C 90.000,E1 46.419} C_DIS
LIN {X 0.061,Y -591.095,Z 1157.051,A 0.000,B 0.000,C 90.000,E1 45.081} C_DIS
LIN {X -0.054,Y -590.746,Z 1157.045,A 0.000,B 0.000,C 90.000,E1 44.028} C_DIS
LIN {X 0.251,Y -590.121,Z 1157.039,A 0.000,B 0.000,C 90.000,E1 42.933} C_DIS
LIN {X -0.040,Y -589.602,Z 1157.034,A 0.000,B 0.000,C 90.000,E1 42.162} C_DIS
LIN {X 0.247,Y -588.647,Z 1157.028,A 0.000,B 0.000,C 90.000,E1 41.067} C_DIS
LIN {X 0.128,Y -587.463,Z 1157.022,A 0.000,B 0.000,C 90.000,E1 40.011} C_DIS
LIN {X 0.254,Y -586.526,Z 1157.018,A 0.000,B 0.000,C 90.000,E1 39.197} C_DIS
LIN {X -0.265,Y -585.111,Z 1157.012,A 0.000,B 0.000,C 90.000,E1 38.177} C_DIS
LIN {X 0.198,Y -582.983,Z 1157.005,A 0.000,B 0.000,C 90.000,E1 36.790} C_DIS
LIN {X -0.073,Y -580.195,Z 1156.997,A 0.000,B 0.000,C 90.000,E1 35.471} C_DIS
LIN {X -0.046,Y -578.139,Z 1156.993,A 0.000,B 0.000,C 90.000,E1 34.659} C_DIS
LIN {X -0.055,Y -576.679,Z 1156.990,A 0.000,B 0.000,C 90.000,E1 34.119} C_DIS
LIN {X 0.076,Y -574.101,Z 1156.985,A 0.000,B 0.000,C 90.000,E1 33.293} C_DIS
LIN {X 0.044,Y -572.220,Z 1156.982,A 0.000,B 0.000,C 90.000,E1 32.752} C_DIS
LIN {X -0.055,Y -568.028,Z 1156.976,A 0.000,B 0.000,C 90.000,E1 31.671} C_DIS
LIN {X -0.123,Y -563.633,Z 1156.971,A 0.000,B 0.000,C 90.000,E1 30.718} C_DIS
LIN {X 0.070,Y -561.626,Z 1156.968,A 0.000,B 0.000,C 90.000,E1 30.285} C_DIS
LIN {X -0.088,Y -556.556,Z 1156.963,A 0.000,B 0.000,C 90.000,E1 29.333} C_DIS
LIN {X 0.124,Y -552.622,Z 1156.959,A 0.000,B 0.000,C 90.000,E1 28.615} C_DIS
LIN {X 0.298,Y -548.320,Z 1156.955,A 0.000,B 0.000,C 90.000,E1 27.897} C_DIS
LIN {X -0.060,Y -545.583,Z 1156.953,A 0.000,B 0.000,C 90.000,E1 27.513} C_DIS
LIN {X -0.071,Y -541.674,Z 1156.950,A 0.000,B 0.000,C 90.000,E1 26.950} C_DIS
LIN {X 0.002,Y -536.444,Z 1156.946,A 0.000,B 0.000,C 90.000,E1 26.232} C_DIS
LIN {X 0.073,Y -533.135,Z 1156.943,A 0.000,B 0.000,C 90.000,E1 25.796} C_DIS
LIN {X -0.090,Y -526.138,Z 1156.939,A 0.000,B 0.000,C 90.000,E1 24.951} C_DIS
LIN {X 0.068,Y -518.633,Z 1156.934,A 0.000,B 0.000,C 90.000,E1 24.079} C_DIS
LIN {X -0.047,Y -513.341,Z 1156.931,A 0.000,B 0.000,C 90.000,E1 23.515} C_DIS
LIN {X 0.242,Y -505.223,Z 1156.926,A 0.000,B 0.000,C 90.000,E1 22.642} C_DIS
LIN {X 0.148,Y -499.587,Z 1156.923,A 0.000,B 0.000,C 90.000,E1 22.099} C_DIS
LIN {X -0.140,Y -492.562,Z 1156.919,A 0.000,B 0.000,C 90.000,E1 21.461} C_DIS
LIN {X -0.135,Y -482.723,Z 1156.914,A 0.000,B 0.000,C 90.000,E1 20.556} C_DIS
LIN {X -0.107,Y -472.482,Z 1156.909,A 0.000,B 0.000,C 90.000,E1 19.631} C_DIS
LIN {X 0.055,Y -465.200,Z 1156.905,A 0.000,B 0.000,C 90.000,E1 18.960} C_DIS
LIN {X -0.062,Y -452.301,Z 1156.899,A 0.000,B 0.000,C 90.000,E1 17.819} C_DIS
LIN {X 0.128,Y -433.337,Z 1156.889,A 0.000,B 0.000,C 90.000,E1 15.969} C_DIS
LIN {X -0.052,Y -420.758,Z 1156.881,A 0.000,B 0.000,C 90.000,E1 14.647} C_DIS
LIN {X 0.065,Y -409.916,Z 1156.874,A 0.000,B 0.000,C 90.000,E1 13.355} C_DIS
LIN {X 0.003,Y -402.261,Z 1156.869,A 0.000,B 0.000,C 90.000,E1 12.355} C_DIS
LIN {X 0.055,Y -397.593,Z 1156.865,A 0.000,B 0.000,C 90.000,E1 11.658} C_DIS
LIN {X 0.125,Y -394.624,Z 1156.862,A 0.000,B 0.000,C 90.000,E1 11.130} C_DIS
LIN {X -0.122,Y -392.770,Z 1156.859,A 0.000,B 0.000,C 90.000,E1 10.658} C_DIS
LIN {X -0.157,Y -392.766,Z 1156.859,A 0.000,B 0.000,C 90.000,E1 10.658} C_DIS
LIN {X -0.066,Y -392.517,Z 1156.857,A 0.000,B 0.000,C 90.000,E1 10.254} C_DIS
LIN {X -0.077,Y -393.260,Z 1156.854,A 0.000,B 0.000,C 90.000,E1 9.726} C_DIS
LIN {X -0.120,Y -394.088,Z 1156.852,A 0.000,B 0.000,C 90.000,E1 9.378} C_DIS
LIN {X 0.158,Y -397.283,Z 1156.846,A 0.000,B 0.000,C 90.000,E1 8.276} C_DIS
LIN {X -0.001,Y -401.651,Z 1156.839,A 0.000,B 0.000,C 90.000,E1 7.068} C_DIS
LIN {X 0.016,Y -402.404,Z 1156.838,A 0.000,B 0.000,C 90.000,E1 6.891} C_DIS
LIN {X 0.104,Y -406.421,Z 1156.834,A 0.000,B 0.000,C 90.000,E1 6.144} C_DIS
LIN {X 0.127,Y -407.665,Z 1156.833,A 0.000,B 0.000,C 90.000,E1 5.967} C_DIS
LIN {X -0.102,Y -412.341,Z 1156.831,A 0.000,B 0.000,C 90.000,E1 5.511} C_DIS
LIN {X -0.062,Y -433.783,Z 1156.822,A 0.000,B 0.000,C 90.000,E1 3.898} C_DIS
LIN {X -0.132,Y -451.556,Z 1156.815,A 0.000,B 0.000,C 90.000,E1 2.636} C_DIS
LIN {X 0.175,Y -466.153,Z 1156.809,A 0.000,B 0.000,C 90.000,E1 1.604} C_DIS
LIN {X 0.189,Y -478.572,Z 1156.804,A 0.000,B 0.000,C 90.000,E1 0.745} C_DIS
LIN {X 0.000,Y -488.910,Z 1156.800,A 0.000,B 0.000,C 90.000,E1 360.000} C_DIS
LIN {X 0.047,Y -496.081,Z 1156.797,A 0.000,B 0.000,C 90.000,E1 359.427} C_DIS
LIN {X 0.201,Y -503.231,Z 1156.793,A 0.000,B 0.000,C 90.000,E1 358.797} C_DIS
LIN {X 0.032,Y -510.128,Z 1156.790,A 0.000,B 0.000,C 90.000,E1 358.165} C_DIS
LIN {X 0.182,Y -516.556,Z 1156.786,A 0.000,B 0.000,C 90.000,E1 357.478} C_DIS
LIN {X -0.031,Y -522.926,Z 1156.782,A 0.000,B 0.000,C 90.000,E1 356.788} C_DIS
LIN {X -0.030,Y -527.674,Z 1156.779,A 0.000,B 0.000,C 90.000,E1 356.216} C_DIS
LIN {X 0.248,Y -533.079,Z 1156.775,A 0.000,B 0.000,C 90.000,E1 355.469} C_DIS
LIN {X -0.006,Y -537.883,Z 1156.771,A 0.000,B 0.000,C 90.000,E1 354.780} C_DIS
LIN {X -0.224,Y -542.250,Z 1156.767,A 0.000,B 0.000,C 90.000,E1 354.090} C_DIS
LIN {X -0.144,Y -545.454,Z 1156.764,A 0.000,B 0.000,C 90.000,E1 353.514} C_DIS
LIN {X 0.051,Y -549.769,Z 1156.759,A 0.000,B 0.000,C 90.000,E1 352.648} C_DIS
LIN {X 0.006,Y -553.006,Z 1156.755,A 0.000,B 0.000,C 90.000,E1 351.951} C_DIS
LIN {X -0.011,Y -555.897,Z 1156.751,A 0.000,B 0.000,C 90.000,E1 351.254} C_DIS
LIN {X -0.254,Y -559.033,Z 1156.747,A 0.000,B 0.000,C 90.000,E1 350.443} C_DIS
LIN {X 0.032,Y -560.978,Z 1156.744,A 0.000,B 0.000,C 90.000,E1 349.859} C_DIS
LIN {X -0.009,Y -564.462,Z 1156.738,A 0.000,B 0.000,C 90.000,E1 348.757} C_DIS
LIN {X -0.067,Y -566.848,Z 1156.733,A 0.000,B 0.000,C 90.000,E1 347.937} C_DIS
LIN {X 0.080,Y -569.792,Z 1156.727,A 0.000,B 0.000,C 90.000,E1 346.825} C_DIS
LIN {X 0.036,Y -573.281,Z 1156.719,A 0.000,B 0.000,C 90.000,E1 345.463} C_DIS
LIN {X 0.213,Y -575.251,Z 1156.715,A 0.000,B 0.000,C 90.000,E1 344.629} C_DIS
LIN {X 0.061,Y -577.769,Z 1156.709,A 0.000,B 0.000,C 90.000,E1 343.559} C_DIS
LIN {X -0.063,Y -580.187,Z 1156.703,A 0.000,B 0.000,C 90.000,E1 342.489} C_DIS
LIN {X -0.139,Y -583.044,Z 1156.695,A 0.000,B 0.000,C 90.000,E1 341.148} C_DIS
LIN {X -0.154,Y -585.559,Z 1156.688,A 0.000,B 0.000,C 90.000,E1 339.806} C_DIS
LIN {X -0.004,Y -587.296,Z 1156.682,A 0.000,B 0.000,C 90.000,E1 338.720} C_DIS
LIN {X -0.049,Y -588.464,Z 1156.677,A 0.000,B 0.000,C 90.000,E1 337.922} C_DIS
LIN {X 0.143,Y -589.326,Z 1156.673,A 0.000,B 0.000,C 90.000,E1 337.102} C_DIS
LIN {X 0.115,Y -590.050,Z 1156.668,A 0.000,B 0.000,C 90.000,E1 336.305} C_DIS
LIN {X -0.209,Y -590.493,Z 1156.664,A 0.000,B 0.000,C 90.000,E1 335.537} C_DIS
LIN {X 0.013,Y -590.648,Z 1156.660,A 0.000,B 0.000,C 90.000,E1 334.717} C_DIS
LIN {X 0.236,Y -590.546,Z 1156.655,A 0.000,B 0.000,C 90.000,E1 333.896} C_DIS
LIN {X -0.180,Y -589.803,Z 1156.649,A 0.000,B 0.000,C 90.000,E1 332.871} C_DIS
LIN {X 0.129,Y -589.197,Z 1156.646,A 0.000,B 0.000,C 90.000,E1 332.308} C_DIS
LIN {X 0.076,Y -587.981,Z 1156.642,A 0.000,B 0.000,C 90.000,E1 331.513} C_DIS
LIN {X 0.018,Y -586.347,Z 1156.637,A 0.000,B 0.000,C 90.000,E1 330.717} C_DIS
LIN {X -0.054,Y -584.284,Z 1156.633,A 0.000,B 0.000,C 90.000,E1 329.921} C_DIS
LIN {X -0.145,Y -581.741,Z 1156.628,A 0.000,B 0.000,C 90.000,E1 329.125} C_DIS
LIN {X -0.281,Y -580.818,Z 1156.627,A 0.000,B 0.000,C 90.000,E1 328.869} C_DIS
LIN {X -0.263,Y -578.706,Z 1156.624,A 0.000,B 0.000,C 90.000,E1 328.329} C_DIS
LIN {X -0.260,Y -576.168,Z 1156.621,A 0.000,B 0.000,C 90.000,E1 327.788} C_DIS
LIN {X -0.194,Y -574.064,Z 1156.619,A 0.000,B 0.000,C 90.000,E1 327.375} C_DIS
LIN {X -0.226,Y -570.810,Z 1156.616,A 0.000,B 0.000,C 90.000,E1 326.834} C_DIS
LIN {X -0.063,Y -566.372,Z 1156.612,A 0.000,B 0.000,C 90.000,E1 326.135} C_DIS
LIN {X -0.152,Y -562.503,Z 1156.609,A 0.000,B 0.000,C 90.000,E1 325.595} C_DIS
LIN {X -0.134,Y -556.072,Z 1156.604,A 0.000,B 0.000,C 90.000,E1 324.769} C_DIS
LIN {X 0.154,Y -547.828,Z 1156.599,A 0.000,B 0.000,C 90.000,E1 323.783} C_DIS
LIN {X -0.275,Y -541.513,Z 1156.595,A 0.000,B 0.000,C 90.000,E1 323.130} C_DIS
LIN {X 0.021,Y -531.196,Z 1156.589,A 0.000,B 0.000,C 90.000,E1 321.984} C_DIS
LIN {X 0.017,Y -528.702,Z 1156.587,A 0.000,B 0.000,C 90.000,E1 321.698} C_DIS
LIN {X 0.092,Y -524.848,Z 1156.584,A 0.000,B 0.000,C 90.000,E1 321.170} C_DIS
LIN {X -0.071,Y -522.854,Z 1156.583,A 0.000,B 0.000,C 90.000,E1 320.848} C_DIS
LIN {X 0.010,Y -520.593,Z 1156.579,A 0.000,B 0.000,C 90.000,E1 320.231} C_DIS
LIN {X 0.058,Y -519.750,Z 1156.576,A 0.000,B 0.000,C 90.000,E1 319.747} C_DIS
LIN {X -0.058,Y -519.401,Z 1156.573,A 0.000,B 0.000,C 90.000,E1 319.175} C_DIS
LIN {X -0.295,Y -519.331,Z 1156.568,A 0.000,B 0.000,C 90.000,E1 318.324} C_DIS
LIN {X 0.100,Y -520.399,Z 1156.554,A 0.000,B 0.000,C 90.000,E1 315.648} C_DIS
LIN {X 0.086,Y -521.124,Z 1156.546,A 0.000,B 0.000,C 90.000,E1 314.190} C_DIS
LIN {X -0.280,Y -521.774,Z 1156.537,A 0.000,B 0.000,C 90.000,E1 312.771} C_DIS
LIN {X -0.248,Y -522.538,Z 1156.529,A 0.000,B 0.000,C 90.000,E1 311.310} C_DIS
LIN {X -0.254,Y -523.456,Z 1156.520,A 0.000,B 0.000,C 90.000,E1 309.564} C_DIS
LIN {X -0.244,Y -524.841,Z 1156.507,A 0.000,B 0.000,C 90.000,E1 307.237} C_DIS
LIN {X 0.351,Y -525.576,Z 1156.500,A 0.000,B 0.000,C 90.000,E1 306.011} C_DIS
LIN {X -0.151,Y -526.580,Z 1156.491,A 0.000,B 0.000,C 90.000,E1 304.326} C_DIS
LIN {X -0.109,Y -528.080,Z 1156.478,A 0.000,B 0.000,C 90.000,E1 302.005} C_DIS
LIN {X -0.078,Y -528.823,Z 1156.471,A 0.000,B 0.000,C 90.000,E1 300.846} C_DIS
LIN {X -0.155,Y -529.751,Z 1156.463,A 0.000,B 0.000,C 90.000,E1 299.411} C_DIS
LIN {X -0.079,Y -530.194,Z 1156.458,A 0.000,B 0.000,C 90.000,E1 298.537} C_DIS
LIN {X -0.082,Y -530.674,Z 1156.452,A 0.000,B 0.000,C 90.000,E1 297.385} C_DIS
LIN {X 0.110,Y -530.981,Z 1156.444,A 0.000,B 0.000,C 90.000,E1 295.924} C_DIS
LIN {X 0.017,Y -531.093,Z 1156.435,A 0.000,B 0.000,C 90.000,E1 294.207} C_DIS
LIN {X 0.188,Y -531.033,Z 1156.425,A 0.000,B 0.000,C 90.000,E1 292.461} C_DIS
LIN {X 0.157,Y -530.983,Z 1156.415,A 0.000,B 0.000,C 90.000,E1 290.737} C_DIS
LIN {X -0.062,Y -530.560,Z 1156.406,A 0.000,B 0.000,C 90.000,E1 289.033} C_DIS
LIN {X 0.007,Y -530.139,Z 1156.399,A 0.000,B 0.000,C 90.000,E1 287.873} C_DIS
LIN {X -0.079,Y -529.570,Z 1156.391,A 0.000,B 0.000,C 90.000,E1 286.441} C_DIS
LIN {X -0.173,Y -528.868,Z 1156.383,A 0.000,B 0.000,C 90.000,E1 285.009} C_DIS
LIN {X 0.096,Y -528.152,Z 1156.375,A 0.000,B 0.000,C 90.000,E1 283.536} C_DIS
LIN {X -0.191,Y -527.447,Z 1156.369,A 0.000,B 0.000,C 90.000,E1 282.411} C_DIS
LIN {X -0.066,Y -526.522,Z 1156.361,A 0.000,B 0.000,C 90.000,E1 280.950} C_DIS
LIN {X 0.002,Y -525.078,Z 1156.348,A 0.000,B 0.000,C 90.000,E1 278.624} C_DIS
LIN {X -0.075,Y -523.998,Z 1156.338,A 0.000,B 0.000,C 90.000,E1 276.891} C_DIS
LIN {X 0.237,Y -522.956,Z 1156.327,A 0.000,B 0.000,C 90.000,E1 274.821} C_DIS
LIN {X 0.071,Y -522.306,Z 1156.319,A 0.000,B 0.000,C 90.000,E1 273.383} C_DIS
LIN {X -0.169,Y -521.650,Z 1156.309,A 0.000,B 0.000,C 90.000,E1 271.661} C_DIS
LIN {X 0.113,Y -521.034,Z 1156.301,A 0.000,B 0.000,C 90.000,E1 270.172} C_DIS
LIN {X -0.188,Y -520.263,Z 1156.291,A 0.000,B 0.000,C 90.000,E1 268.453} C_DIS
LIN {X 0.048,Y -519.477,Z 1156.282,A 0.000,B 0.000,C 90.000,E1 266.674} C_DIS
LIN {X -0.158,Y -518.752,Z 1156.275,A 0.000,B 0.000,C 90.000,E1 265.527} C_DIS
LIN {X 0.180,Y -517.926,Z 1156.269,A 0.000,B 0.000,C 90.000,E1 264.318} C_DIS
LIN {X -0.135,Y -515.950,Z 1156.257,A 0.000,B 0.000,C 90.000,E1 262.299} C_DIS
LIN {X 0.156,Y -513.913,Z 1156.246,A 0.000,B 0.000,C 90.000,E1 260.208} C_DIS
LIN {X -0.117,Y -511.914,Z 1156.234,A 0.000,B 0.000,C 90.000,E1 258.173} C_DIS
LIN {X -0.240,Y -510.074,Z 1156.223,A 0.000,B 0.000,C 90.000,E1 256.117} C_DIS
LIN {X -0.153,Y -508.279,Z 1156.211,A 0.000,B 0.000,C 90.000,E1 254.031} C_DIS
LIN {X -0.050,Y -506.652,Z 1156.201,A 0.000,B 0.000,C 90.000,E1 252.236} C_DIS
LIN {X 0.167,Y -504.909,Z 1156.191,A 0.000,B 0.000,C 90.000,E1 250.423} C_DIS
LIN {X -0.046,Y -503.430,Z 1156.183,A 0.000,B 0.000,C 90.000,E1 248.954} C_DIS
LIN {X -0.290,Y -501.989,Z 1156.175,A 0.000,B 0.000,C 90.000,E1 247.486} C_DIS
LIN {X -0.106,Y -499.867,Z 1156.165,A 0.000,B 0.000,C 90.000,E1 245.665} C_DIS
LIN {X -0.088,Y -498.322,Z 1156.158,A 0.000,B 0.000,C 90.000,E1 244.460} C_DIS
LIN {X 0.222,Y -495.863,Z 1156.148,A 0.000,B 0.000,C 90.000,E1 242.615} C_DIS
LIN {X -0.155,Y -492.819,Z 1156.136,A 0.000,B 0.000,C 90.000,E1 240.539} C_DIS
LIN {X -0.047,Y -491.454,Z 1156.131,A 0.000,B 0.000,C 90.000,E1 239.616} C_DIS
LIN {X 0.122,Y -489.158,Z 1156.123,A 0.000,B 0.000,C 90.000,E1 238.074} C_DIS
LIN {X -0.282,Y -485.382,Z 1156.109,A 0.000,B 0.000,C 90.000,E1 235.674} C_DIS
LIN {X 0.120,Y -482.573,Z 1156.099,A 0.000,B 0.000,C 90.000,E1 233.783} C_DIS
LIN {X 0.058,Y -480.642,Z 1156.092,A 0.000,B 0.000,C 90.000,E1 232.557} C_DIS
LIN {X -0.023,Y -477.205,Z 1156.080,A 0.000,B 0.000,C 90.000,E1 230.400} C_DIS
LIN {X 0.024,Y -474.256,Z 1156.070,A 0.000,B 0.000,C 90.000,E1 228.528} C_DIS
LIN {X -0.133,Y -471.661,Z 1156.061,A 0.000,B 0.000,C 90.000,E1 226.986} C_DIS
LIN {X -0.020,Y -469.128,Z 1156.052,A 0.000,B 0.000,C 90.000,E1 225.405} C_DIS
LIN {X 0.188,Y -464.245,Z 1156.031,A 0.000,B 0.000,C 90.000,E1 221.595} C_DIS
LIN {X 0.088,Y -462.100,Z 1156.017,A 0.000,B 0.000,C 90.000,E1 219.072} C_DIS
LIN {X -0.240,Y -461.030,Z 1156.008,A 0.000,B 0.000,C 90.000,E1 217.523} C_DIS
LIN {X 0.005,Y -459.520,Z 1155.994,A 0.000,B 0.000,C 90.000,E1 214.945} C_DIS
LIN {X -0.241,Y -458.716,Z 1155.975,A 0.000,B 0.000,C 90.000,E1 211.465} C_DIS
LIN {X -0.241,Y -460.984,Z 1155.946,A 0.000,B 0.000,C 90.000,E1 206.360} C_DIS
LIN {X 0.137,Y -463.911,Z 1155.932,A 0.000,B 0.000,C 90.000,E1 203.770} C_DIS
LIN {X 0.097,Y -470.141,Z 1155.913,A 0.000,B 0.000,C 90.000,E1 200.301} C_DIS
LIN {X -0.054,Y -475.424,Z 1155.901,A 0.000,B 0.000,C 90.000,E1 198.127} C_DIS
LIN {X -0.216,Y -482.599,Z 1155.887,A 0.000,B 0.000,C 90.000,E1 195.662} C_DIS
LIN {X 0.043,Y -489.717,Z 1155.875,A 0.000,B 0.000,C 90.000,E1 193.480} C_DIS
LIN {X -0.087,Y -496.940,Z 1155.863,A 0.000,B 0.000,C 90.000,E1 191.366} C_DIS
LIN {X 0.003,Y -502.404,Z 1155.855,A 0.000,B 0.000,C 90.000,E1 189.849} C_DIS
LIN {X -0.039,Y -511.237,Z 1155.842,A 0.000,B 0.000,C 90.000,E1 187.466} C_DIS
LIN {X 0.158,Y -516.808,Z 1155.833,A 0.000,B 0.000,C 90.000,E1 185.967} C_DIS
LIN {X -0.106,Y -522.248,Z 1155.825,A 0.000,B 0.000,C 90.000,E1 184.531} C_DIS
LIN {X 0.252,Y -527.664,Z 1155.817,A 0.000,B 0.000,C 90.000,E1 183.037} C_DIS
LIN {X 0.153,Y -533.043,Z 1155.809,A 0.000,B 0.000,C 90.000,E1 181.604} C_DIS
LIN {X 0.135,Y -537.370,Z 1155.803,A 0.000,B 0.000,C 90.000,E1 180.458} C_DIS
LIN {X 0.258,Y -544.910,Z 1155.792,A 0.000,B 0.000,C 90.000,E1 178.453} C_DIS
LIN {X 0.006,Y -551.380,Z 1155.782,A 0.000,B 0.000,C 90.000,E1 176.788} C_DIS
LIN {X -0.100,Y -557.872,Z 1155.773,A 0.000,B 0.000,C 90.000,E1 175.122} C_DIS
LIN {X -0.021,Y -564.218,Z 1155.764,A 0.000,B 0.000,C 90.000,E1 173.451} C_DIS
LIN {X 0.091,Y -569.569,Z 1155.756,A 0.000,B 0.000,C 90.000,E1 172.064} C_DIS
LIN {X -0.078,Y -575.862,Z 1155.747,A 0.000,B 0.000,C 90.000,E1 170.443} C_DIS
LIN {X -0.027,Y -582.046,Z 1155.738,A 0.000,B 0.000,C 90.000,E1 168.814} C_DIS
LIN {X -0.227,Y -586.116,Z 1155.732,A 0.000,B 0.000,C 90.000,E1 167.757} C_DIS
LIN {X 0.204,Y -590.043,Z 1155.726,A 0.000,B 0.000,C 90.000,E1 166.645} C_DIS
LIN {X 0.109,Y -593.850,Z 1155.720,A 0.000,B 0.000,C 90.000,E1 165.589} C_DIS
LIN {X -0.083,Y -598.424,Z 1155.713,A 0.000,B 0.000,C 90.000,E1 164.283} C_DIS
LIN {X 0.254,Y -601.957,Z 1155.707,A 0.000,B 0.000,C 90.000,E1 163.196} C_DIS
LIN {X -0.105,Y -605.360,Z 1155.701,A 0.000,B 0.000,C 90.000,E1 162.181} C_DIS
LIN {X -0.236,Y -608.621,Z 1155.695,A 0.000,B 0.000,C 90.000,E1 161.148} C_DIS
LIN {X -0.058,Y -613.262,Z 1155.687,A 0.000,B 0.000,C 90.000,E1 159.571} C_DIS
LIN {X -0.119,Y -616.910,Z 1155.679,A 0.000,B 0.000,C 90.000,E1 158.284} C_DIS
LIN {X -0.141,Y -621.149,Z 1155.671,A 0.000,B 0.000,C 90.000,E1 156.741} C_DIS
LIN {X 0.157,Y -624.503,Z 1155.664,A 0.000,B 0.000,C 90.000,E1 155.433} C_DIS
LIN {X 0.209,Y -627.833,Z 1155.657,A 0.000,B 0.000,C 90.000,E1 154.152} C_DIS
LIN {X -0.176,Y -632.207,Z 1155.647,A 0.000,B 0.000,C 90.000,E1 152.410} C_DIS
LIN {X 0.005,Y -635.175,Z 1155.640,A 0.000,B 0.000,C 90.000,E1 151.129} C_DIS
LIN {X -0.019,Y -637.981,Z 1155.633,A 0.000,B 0.000,C 90.000,E1 149.871} C_DIS
LIN {X 0.002,Y -640.644,Z 1155.626,A 0.000,B 0.000,C 90.000,E1 148.614} C_DIS
LIN {X 0.346,Y -642.621,Z 1155.620,A 0.000,B 0.000,C 90.000,E1 147.582} C_DIS
LIN {X 0.301,Y -645.362,Z 1155.612,A 0.000,B 0.000,C 90.000,E1 146.087} C_DIS
LIN {X -0.293,Y -647.566,Z 1155.605,A 0.000,B 0.000,C 90.000,E1 144.895} C_DIS
LIN {X 0.055,Y -649.709,Z 1155.598,A 0.000,B 0.000,C 90.000,E1 143.623} C_DIS
LIN {X -0.106,Y -652.553,Z 1155.588,A 0.000,B 0.000,C 90.000,E1 141.904} C_DIS
LIN {X 0.195,Y -655.672,Z 1155.579,A 0.000,B 0.000,C 90.000,E1 140.150} C_DIS
LIN {X 0.057,Y -658.106,Z 1155.572,A 0.000,B 0.000,C 90.000,E1 138.933} C_DIS
LIN {X -0.063,Y -661.141,Z 1155.564,A 0.000,B 0.000,C 90.000,E1 137.472} C_DIS
LIN {X 0.324,Y -664.056,Z 1155.556,A 0.000,B 0.000,C 90.000,E1 135.972} C_DIS
LIN {X 0.310,Y -669.312,Z 1155.542,A 0.000,B 0.000,C 90.000,E1 133.542} C_DIS
LIN {X -0.005,Y -673.823,Z 1155.531,A 0.000,B 0.000,C 90.000,E1 131.634} C_DIS
LIN {X 0.377,Y -679.690,Z 1155.518,A 0.000,B 0.000,C 90.000,E1 129.197} C_DIS
LIN {X 0.198,Y -682.735,Z 1155.511,A 0.000,B 0.000,C 90.000,E1 128.016} C_DIS
LIN {X -0.152,Y -686.884,Z 1155.502,A 0.000,B 0.000,C 90.000,E1 126.377} C_DIS
LIN {X 0.285,Y -689.248,Z 1155.497,A 0.000,B 0.000,C 90.000,E1 125.391} C_DIS
LIN {X -0.177,Y -692.132,Z 1155.490,A 0.000,B 0.000,C 90.000,E1 124.246} C_DIS
LIN {X 0.162,Y -694.920,Z 1155.484,A 0.000,B 0.000,C 90.000,E1 123.038} C_DIS
LIN {X 0.076,Y -696.517,Z 1155.480,A 0.000,B 0.000,C 90.000,E1 122.339} C_DIS
LIN {X -0.120,Y -698.454,Z 1155.474,A 0.000,B 0.000,C 90.000,E1 121.416} C_DIS
LIN {X -0.268,Y -700.590,Z 1155.468,A 0.000,B 0.000,C 90.000,E1 120.256} C_DIS
LIN {X 0.141,Y -703.127,Z 1155.460,A 0.000,B 0.000,C 90.000,E1 118.821} C_DIS
LIN {X 0.029,Y -704.689,Z 1155.455,A 0.000,B 0.000,C 90.000,E1 117.897} C_DIS
LIN {X -0.023,Y -705.355,Z 1155.453,A 0.000,B 0.000,C 90.000,E1 117.436} C_DIS
LIN {X -0.104,Y -706.004,Z 1155.449,A 0.000,B 0.000,C 90.000,E1 116.744} C_DIS
LIN {X 0.124,Y -706.504,Z 1155.443,A 0.000,B 0.000,C 90.000,E1 115.796} C_DIS
LIN {X 0.368,Y -706.612,Z 1155.440,A 0.000,B 0.000,C 90.000,E1 115.079} C_DIS
LIN {X 0.016,Y -706.462,Z 1155.437,A 0.000,B 0.000,C 90.000,E1 114.643} C_DIS
LIN {X 0.308,Y -706.158,Z 1155.436,A 0.000,B 0.000,C 90.000,E1 114.387} C_DIS
LIN {X -0.045,Y -705.222,Z 1155.433,A 0.000,B 0.000,C 90.000,E1 113.951} C_DIS
LIN {X 0.245,Y -703.297,Z 1155.431,A 0.000,B 0.000,C 90.000,E1 113.462} C_DIS
LIN {X -0.119,Y -702.108,Z 1155.429,A 0.000,B 0.000,C 90.000,E1 113.259} C_DIS
LIN {X 0.319,Y -697.947,Z 1155.427,A 0.000,B 0.000,C 90.000,E1 112.770} C_DIS
LIN {X -0.195,Y -696.744,Z 1155.426,A 0.000,B 0.000,C 90.000,E1 112.695} C_DIS
LIN {X -0.333,Y -694.953,Z 1155.425,A 0.000,B 0.000,C 90.000,E1 112.589} C_DIS
LIN {X 0.072,Y -692.450,Z 1155.425,A 0.000,B 0.000,C 90.000,E1 112.461} C_DIS
LIN {X 0.414,Y -685.292,Z 1155.424,A 0.000,B 0.000,C 90.000,E1 112.206} C_DIS
LIN {X 0.028,Y -682.298,Z 1155.423,A 0.000,B 0.000,C 90.000,E1 112.206} C_DIS
LIN {X 0.188,Y -676.744,Z 1155.423,A 0.000,B 0.000,C 90.000,E1 112.153} C_DIS
LIN {X 0.120,Y -603.926,Z 1155.423,A 0.000,B 0.000,C 90.000,E1 112.153} C_DIS
LIN {X -0.190,Y -600.678,Z 1155.422,A 0.000,B 0.000,C 90.000,E1 111.972} C_DIS
LIN {X 0.029,Y -593.188,Z 1155.419,A 0.000,B 0.000,C 90.000,E1 111.354} C_DIS
LIN {X 0.067,Y -576.976,Z 1155.411,A 0.000,B 0.000,C 90.000,E1 109.939} C_DIS
LIN {X 0.008,Y -574.138,Z 1155.410,A 0.000,B 0.000,C 90.000,E1 109.704} C_DIS
LIN {X -0.194,Y -568.129,Z 1155.407,A 0.000,B 0.000,C 90.000,E1 109.268} C_DIS
LIN {X -0.060,Y -560.192,Z 1155.404,A 0.000,B 0.000,C 90.000,E1 108.725} C_DIS
LIN {X -0.006,Y -555.497,Z 1155.402,A 0.000,B 0.000,C 90.000,E1 108.417} C_DIS
LIN {X 0.247,Y -551.413,Z 1155.401,A 0.000,B 0.000,C 90.000,E1 108.055} C_DIS
LIN {X 0.026,Y -550.206,Z 1155.399,A 0.000,B 0.000,C 90.000,E1 107.873} C_DIS
LIN {X -0.017,Y -550.189,Z 1155.399,A 0.000,B 0.000,C 90.000,E1 107.873} C_DIS
LIN {X -0.199,Y -549.883,Z 1155.397,A 0.000,B 0.000,C 90.000,E1 107.511} C_DIS
LIN {X -0.155,Y -551.547,Z 1155.384,A 0.000,B 0.000,C 90.000,E1 105.064} C_DIS
LIN {X 0.127,Y -552.935,Z 1155.374,A 0.000,B 0.000,C 90.000,E1 103.355} C_DIS
LIN {X -0.217,Y -554.447,Z 1155.365,A 0.000,B 0.000,C 90.000,E1 101.715} C_DIS
LIN {X -0.119,Y -555.814,Z 1155.357,A 0.000,B 0.000,C 90.000,E1 100.310} C_DIS
LIN {X -0.100,Y -557.122,Z 1155.349,A 0.000,B 0.000,C 90.000,E1 98.916} C_DIS
LIN {X -0.002,Y -558.556,Z 1155.340,A 0.000,B 0.000,C 90.000,E1 97.239} C_DIS
LIN {X 0.193,Y -559.998,Z 1155.329,A 0.000,B 0.000,C 90.000,E1 95.277} C_DIS
LIN {X 0.018,Y -560.834,Z 1155.323,A 0.000,B 0.000,C 90.000,E1 94.188} C_DIS
LIN {X 0.181,Y -562.291,Z 1155.313,A 0.000,B 0.000,C 90.000,E1 92.236} C_DIS
LIN {X 0.141,Y -563.372,Z 1155.305,A 0.000,B 0.000,C 90.000,E1 90.859} C_DIS
LIN {X -0.238,Y -564.749,Z 1155.294,A 0.000,B 0.000,C 90.000,E1 88.969} C_DIS
LIN {X -0.017,Y -565.876,Z 1155.283,A 0.000,B 0.000,C 90.000,E1 87.020} C_DIS
LIN {X -0.263,Y -566.987,Z 1155.273,A 0.000,B 0.000,C 90.000,E1 85.122} C_DIS
LIN {X -0.183,Y -567.848,Z 1155.265,A 0.000,B 0.000,C 90.000,E1 83.742} C_DIS
LIN {X 0.147,Y -568.751,Z 1155.256,A 0.000,B 0.000,C 90.000,E1 82.064} C_DIS
LIN {X 0.132,Y -569.294,Z 1155.250,A 0.000,B 0.000,C 90.000,E1 80.971} C_DIS
LIN {X -0.174,Y -569.936,Z 1155.242,A 0.000,B 0.000,C 90.000,E1 79.634} C_DIS
LIN {X -0.169,Y -570.737,Z 1155.233,A 0.000,B 0.000,C 90.000,E1 77.993} C_DIS
LIN {X -0.147,Y -571.523,Z 1155.224,A 0.000,B 0.000,C 90.000,E1 76.353} C_DIS
LIN {X 0.018,Y -572.348,Z 1155.215,A 0.000,B 0.000,C 90.000,E1 74.700} C_DIS
LIN {X 0.142,Y -573.773,Z 1155.201,A 0.000,B 0.000,C 90.000,E1 72.236} C_DIS
LIN {X -0.229,Y -575.093,Z 1155.191,A 0.000,B 0.000,C 90.000,E1 70.369} C_DIS
LIN {X -0.179,Y -577.206,Z 1155.177,A 0.000,B 0.000,C 90.000,E1 67.922} C_DIS
LIN {X -0.254,Y -578.772,Z 1155.168,A 0.000,B 0.000,C 90.000,E1 66.305} C_DIS
LIN {X -0.060,Y -580.230,Z 1155.159,A 0.000,B 0.000,C 90.000,E1 64.665} C_DIS
LIN {X 0.036,Y -581.494,Z 1155.152,A 0.000,B 0.000,C 90.000,E1 63.307} C_DIS
LIN {X -0.096,Y -583.204,Z 1155.141,A 0.000,B 0.000,C 90.000,E1 61.435} C_DIS
LIN {X 0.211,Y -584.523,Z 1155.132,A 0.000,B 0.000,C 90.000,E1 59.793} C_DIS
LIN {X 0.165,Y -585.532,Z 1155.125,A 0.000,B 0.000,C 90.000,E1 58.456} C_DIS
LIN {X 0.314,Y -586.587,Z 1155.116,A 0.000,B 0.000,C 90.000,E1 56.834} C_DIS
LIN {X -0.069,Y -587.284,Z 1155.110,A 0.000,B 0.000,C 90.000,E1 55.801} C_DIS
LIN {X -0.052,Y -588.264,Z 1155.101,A 0.000,B 0.000,C 90.000,E1 54.196} C_DIS
LIN {X 0.061,Y -589.325,Z 1155.091,A 0.000,B 0.000,C 90.000,E1 52.316} C_DIS
LIN {X -0.210,Y -590.043,Z 1155.083,A 0.000,B 0.000,C 90.000,E1 51.009} C_DIS
LIN {X 0.150,Y -590.485,Z 1155.077,A 0.000,B 0.000,C 90.000,E1 49.908} C_DIS
LIN {X -0.141,Y -590.726,Z 1155.073,A 0.000,B 0.000,C 90.000,E1 49.138} C_DIS
LIN {X -0.028,Y -590.982,Z 1155.066,A 0.000,B 0.000,C 90.000,E1 47.796} C_DIS
LIN {X 0.038,Y -590.982,Z 1155.058,A 0.000,B 0.000,C 90.000,E1 46.458} C_DIS
LIN {X -0.318,Y -590.813,Z 1155.051,A 0.000,B 0.000,C 90.000,E1 45.162} C_DIS
LIN {X 0.400,Y -590.477,Z 1155.045,A 0.000,B 0.000,C 90.000,E1 44.028} C_DIS
LIN {X -0.133,Y -589.840,Z 1155.039,A 0.000,B 0.000,C 90.000,E1 43.014} C_DIS
LIN {X -0.031,Y -589.316,Z 1155.035,A 0.000,B 0.000,C 90.000,E1 42.204} C_DIS
LIN {X -0.142,Y -588.355,Z 1155.029,A 0.000,B 0.000,C 90.000,E1 41.148} C_DIS
LIN {X -0.263,Y -587.171,Z 1155.023,A 0.000,B 0.000,C 90.000,E1 40.092} C_DIS
LIN {X 0.052,Y -585.880,Z 1155.017,A 0.000,B 0.000,C 90.000,E1 38.991} C_DIS
LIN {X 0.162,Y -584.810,Z 1155.012,A 0.000,B 0.000,C 90.000,E1 38.177} C_DIS
LIN {X -0.197,Y -582.633,Z 1155.005,A 0.000,B 0.000,C 90.000,E1 36.870} C_DIS
LIN {X 0.335,Y -580.995,Z 1155.000,A 0.000,B 0.000,C 90.000,E1 36.011} C_DIS
LIN {X 0.035,Y -579.185,Z 1154.996,A 0.000,B 0.000,C 90.000,E1 35.231} C_DIS
LIN {X 0.193,Y -577.033,Z 1154.991,A 0.000,B 0.000,C 90.000,E1 34.405} C_DIS
LIN {X 0.180,Y -575.489,Z 1154.988,A 0.000,B 0.000,C 90.000,E1 33.865} C_DIS
LIN {X -0.320,Y -573.747,Z 1154.985,A 0.000,B 0.000,C 90.000,E1 33.372} C_DIS
LIN {X -0.042,Y -571.852,Z 1154.982,A 0.000,B 0.000,C 90.000,E1 32.801} C_DIS
LIN {X -0.269,Y -568.668,Z 1154.978,A 0.000,B 0.000,C 90.000,E1 32.005} C_DIS
LIN {X -0.152,Y -567.614,Z 1154.976,A 0.000,B 0.000,C 90.000,E1 31.720} C_DIS
LIN {X -0.033,Y -563.226,Z 1154.971,A 0.000,B 0.000,C 90.000,E1 30.747} C_DIS
LIN {X -0.041,Y -561.225,Z 1154.969,A 0.000,B 0.000,C 90.000,E1 30.335} C_DIS
LIN {X 0.279,Y -556.147,Z 1154.963,A 0.000,B 0.000,C 90.000,E1 29.333} C_DIS
LIN {X -0.114,Y -551.347,Z 1154.958,A 0.000,B 0.000,C 90.000,E1 28.537} C_DIS
LIN {X -0.207,Y -546.992,Z 1154.955,A 0.000,B 0.000,C 90.000,E1 27.847} C_DIS
LIN {X -0.209,Y -541.200,Z 1154.950,A 0.000,B 0.000,C 90.000,E1 27.001} C_DIS
LIN {X -0.008,Y -537.075,Z 1154.947,A 0.000,B 0.000,C 90.000,E1 26.411} C_DIS
LIN {X 0.064,Y -533.843,Z 1154.944,A 0.000,B 0.000,C 90.000,E1 25.976} C_DIS
LIN {X -0.318,Y -526.818,Z 1154.940,A 0.000,B 0.000,C 90.000,E1 25.155} C_DIS
LIN {X 0.025,Y -519.397,Z 1154.935,A 0.000,B 0.000,C 90.000,E1 24.259} C_DIS
LIN {X -0.136,Y -514.134,Z 1154.932,A 0.000,B 0.000,C 90.000,E1 23.695} C_DIS
LIN {X 0.043,Y -505.985,Z 1154.927,A 0.000,B 0.000,C 90.000,E1 22.823} C_DIS
LIN {X -0.141,Y -498.934,Z 1154.923,A 0.000,B 0.000,C 90.000,E1 22.153} C_DIS
LIN {X 0.033,Y -491.925,Z 1154.919,A 0.000,B 0.000,C 90.000,E1 21.461} C_DIS
LIN {X -0.024,Y -481.980,Z 1154.914,A 0.000,B 0.000,C 90.000,E1 20.556} C_DIS
LIN {X -0.011,Y -470.247,Z 1154.908,A 0.000,B 0.000,C 90.000,E1 19.504} C_DIS
LIN {X 0.239,Y -464.498,Z 1154.906,A 0.000,B 0.000,C 90.000,E1 18.960} C_DIS
LIN {X 0.045,Y -441.389,Z 1154.894,A 0.000,B 0.000,C 90.000,E1 16.858} C_DIS
LIN {X -0.042,Y -427.083,Z 1154.886,A 0.000,B 0.000,C 90.000,E1 15.426} C_DIS
LIN {X 0.165,Y -413.208,Z 1154.877,A 0.000,B 0.000,C 90.000,E1 13.828} C_DIS
LIN {X 0.094,Y -405.205,Z 1154.871,A 0.000,B 0.000,C 90.000,E1 12.827} C_DIS
LIN {X -0.167,Y -399.116,Z 1154.867,A 0.000,B 0.000,C 90.000,E1 12.007} C_DIS
LIN {X -0.148,Y -395.882,Z 1154.864,A 0.000,B 0.000,C 90.000,E1 11.478} C_DIS
LIN {X 0.102,Y -394.264,Z 1154.862,A 0.000,B 0.000,C 90.000,E1 11.130} C_DIS
LIN {X -0.066,Y -392.621,Z 1154.859,A 0.000,B 0.000,C 90.000,E1 10.658} C_DIS
LIN {X -0.104,Y -392.614,Z 1154.859,A 0.000,B 0.000,C 90.000,E1 10.658} C_DIS
LIN {X -0.210,Y -392.551,Z 1154.857,A 0.000,B 0.000,C 90.000,E1 10.197} C_DIS
LIN {X -0.074,Y -393.609,Z 1154.853,A 0.000,B 0.000,C 90.000,E1 9.557} C_DIS
LIN {X -0.076,Y -396.650,Z 1154.847,A 0.000,B 0.000,C 90.000,E1 8.511} C_DIS
LIN {X 0.171,Y -401.532,Z 1154.839,A 0.000,B 0.000,C 90.000,E1 7.068} C_DIS
LIN {X 0.160,Y -403.094,Z 1154.838,A 0.000,B 0.000,C 90.000,E1 6.720} C_DIS
LIN {X -0.063,Y -406.319,Z 1154.834,A 0.000,B 0.000,C 90.000,E1 6.144} C_DIS
LIN {X -0.094,Y -407.098,Z 1154.833,A 0.000,B 0.000,C 90.000,E1 6.024} C_DIS
LIN {X 0.130,Y -410.924,Z 1154.831,A 0.000,B 0.000,C 90.000,E1 5.568} C_DIS
LIN {X -0.158,Y -412.613,Z 1154.830,A 0.000,B 0.000,C 90.000,E1 5.448} C_DIS
LIN {X -0.169,Y -435.659,Z 1154.821,A 0.000,B 0.000,C 90.000,E1 3.726} C_DIS
LIN {X -0.107,Y -456.723,Z 1154.812,A 0.000,B 0.000,C 90.000,E1 2.236} C_DIS
LIN {X 0.181,Y -468.028,Z 1154.808,A 0.000,B 0.000,C 90.000,E1 1.432} C_DIS
LIN {X -0.143,Y -476.174,Z 1154.805,A 0.000,B 0.000,C 90.000,E1 0.917} C_DIS
LIN {X 0.048,Y -485.311,Z 1154.801,A 0.000,B 0.000,C 90.000,E1 0.229} C_DIS
LIN {X 0.154,Y -492.662,Z 1154.798,A 0.000,B 0.000,C 90.000,E1 359.656} C_DIS
LIN {X 0.033,Y -497.135,Z 1154.796,A 0.000,B 0.000,C 90.000,E1 359.312} C_DIS
LIN {X 0.184,Y -502.976,Z 1154.793,A 0.000,B 0.000,C 90.000,E1 358.797} C_DIS
LIN {X -0.258,Y -509.696,Z 1154.790,A 0.000,B 0.000,C 90.000,E1 358.224} C_DIS
LIN {X -0.237,Y -516.363,Z 1154.786,A 0.000,B 0.000,C 90.000,E1 357.535} C_DIS
LIN {X -0.176,Y -522.550,Z 1154.782,A 0.000,B 0.000,C 90.000,E1 356.846} C_DIS
LIN {X -0.222,Y -527.384,Z 1154.779,A 0.000,B 0.000,C 90.000,E1 356.274} C_DIS
LIN {X -0.001,Y -532.905,Z 1154.775,A 0.000,B 0.000,C 90.000,E1 355.527} C_DIS
LIN {X -0.258,Y -537.793,Z 1154.771,A 0.000,B 0.000,C 90.000,E1 354.837} C_DIS
LIN {X 0.061,Y -542.208,Z 1154.767,A 0.000,B 0.000,C 90.000,E1 354.090} C_DIS
LIN {X 0.142,Y -545.465,Z 1154.764,A 0.000,B 0.000,C 90.000,E1 353.514} C_DIS
LIN {X -0.206,Y -549.783,Z 1154.759,A 0.000,B 0.000,C 90.000,E1 352.704} C_DIS
LIN {X -0.072,Y -552.473,Z 1154.756,A 0.000,B 0.000,C 90.000,E1 352.129} C_DIS
LIN {X 0.159,Y -554.902,Z 1154.753,A 0.000,B 0.000,C 90.000,E1 351.546} C_DIS
LIN {X -0.095,Y -558.137,Z 1154.749,A 0.000,B 0.000,C 90.000,E1 350.735} C_DIS
LIN {X -0.224,Y -561.150,Z 1154.744,A 0.000,B 0.000,C 90.000,E1 349.916} C_DIS
LIN {X -0.260,Y -564.658,Z 1154.738,A 0.000,B 0.000,C 90.000,E1 348.814} C_DIS
LIN {X 0.239,Y -567.097,Z 1154.733,A 0.000,B 0.000,C 90.000,E1 347.937} C_DIS
LIN {X 0.018,Y -570.767,Z 1154.726,A 0.000,B 0.000,C 90.000,E1 346.589} C_DIS
LIN {X -0.009,Y -574.251,Z 1154.718,A 0.000,B 0.000,C 90.000,E1 345.227} C_DIS
LIN {X -0.167,Y -578.112,Z 1154.709,A 0.000,B 0.000,C 90.000,E1 343.614} C_DIS
LIN {X 0.100,Y -581.123,Z 1154.701,A 0.000,B 0.000,C 90.000,E1 342.236} C_DIS
LIN {X 0.201,Y -583.430,Z 1154.695,A 0.000,B 0.000,C 90.000,E1 341.148} C_DIS
LIN {X -0.218,Y -585.474,Z 1154.689,A 0.000,B 0.000,C 90.000,E1 340.115} C_DIS
LIN {X 0.273,Y -586.885,Z 1154.685,A 0.000,B 0.000,C 90.000,E1 339.263} C_DIS
LIN {X -0.112,Y -588.566,Z 1154.679,A 0.000,B 0.000,C 90.000,E1 338.230} C_DIS
LIN {X 0.080,Y -589.591,Z 1154.675,A 0.000,B 0.000,C 90.000,E1 337.411} C_DIS
LIN {X -0.053,Y -590.567,Z 1154.669,A 0.000,B 0.000,C 90.000,E1 336.357} C_DIS
LIN {X 0.066,Y -591.178,Z 1154.663,A 0.000,B 0.000,C 90.000,E1 335.281} C_DIS
LIN {X 0.196,Y -591.265,Z 1154.657,A 0.000,B 0.000,C 90.000,E1 334.204} C_DIS
LIN {X -0.004,Y -591.096,Z 1154.654,A 0.000,B 0.000,C 90.000,E1 333.691} C_DIS
LIN {X 0.219,Y -590.500,Z 1154.649,A 0.000,B 0.000,C 90.000,E1 332.871} C_DIS
LIN {X 0.011,Y -589.929,Z 1154.646,A 0.000,B 0.000,C 90.000,E1 332.359} C_DIS
LIN {X -0.030,Y -588.794,Z 1154.642,A 0.000,B 0.000,C 90.000,E1 331.563} C_DIS
LIN {X -0.363,Y -587.232,Z 1154.638,A 0.000,B 0.000,C 90.000,E1 330.795} C_DIS
LIN {X 0.201,Y -585.952,Z 1154.635,A 0.000,B 0.000,C 90.000,E1 330.205} C_DIS
LIN {X 0.249,Y -584.522,Z 1154.632,A 0.000,B 0.000,C 90.000,E1 329.665} C_DIS
LIN {X 0.156,Y -581.931,Z 1154.627,A 0.000,B 0.000,C 90.000,E1 328.869} C_DIS
LIN {X 0.033,Y -578.725,Z 1154.623,A 0.000,B 0.000,C 90.000,E1 328.074} C_DIS
LIN {X 0.259,Y -575.389,Z 1154.619,A 0.000,B 0.000,C 90.000,E1 327.375} C_DIS
LIN {X 0.147,Y -571.372,Z 1154.615,A 0.000,B 0.000,C 90.000,E1 326.707} C_DIS
LIN {X 0.309,Y -566.937,Z 1154.611,A 0.000,B 0.000,C 90.000,E1 326.008} C_DIS
LIN {X 0.219,Y -563.071,Z 1154.608,A 0.000,B 0.000,C 90.000,E1 325.468} C_DIS
LIN {X -0.149,Y -557.735,Z 1154.604,A 0.000,B 0.000,C 90.000,E1 324.815} C_DIS
LIN {X 0.162,Y -549.586,Z 1154.599,A 0.000,B 0.000,C 90.000,E1 323.829} C_DIS
LIN {X 0.150,Y -543.248,Z 1154.595,A 0.000,B 0.000,C 90.000,E1 323.130} C_DIS
LIN {X 0.271,Y -529.489,Z 1154.587,A 0.000,B 0.000,C 90.000,E1 321.618} C_DIS
LIN {X 0.068,Y -525.570,Z 1154.584,A 0.000,B 0.000,C 90.000,E1 321.126} C_DIS
LIN {X -0.221,Y -523.120,Z 1154.582,A 0.000,B 0.000,C 90.000,E1 320.723} C_DIS
LIN {X 0.023,Y -521.365,Z 1154.579,A 0.000,B 0.000,C 90.000,E1 320.231} C_DIS
LIN {X 0.166,Y -520.923,Z 1154.578,A 0.000,B 0.000,C 90.000,E1 320.070} C_DIS
LIN {X 0.000,Y -519.976,Z 1154.575,A 0.000,B 0.000,C 90.000,E1 319.504} C_DIS
LIN {X -0.036,Y -519.676,Z 1154.569,A 0.000,B 0.000,C 90.000,E1 318.485} C_DIS
LIN {X -0.079,Y -520.709,Z 1154.553,A 0.000,B 0.000,C 90.000,E1 315.567} C_DIS
LIN {X -0.017,Y -521.298,Z 1154.547,A 0.000,B 0.000,C 90.000,E1 314.393} C_DIS
LIN {X 0.056,Y -521.803,Z 1154.540,A 0.000,B 0.000,C 90.000,E1 313.218} C_DIS
LIN {X 0.030,Y -522.640,Z 1154.531,A 0.000,B 0.000,C 90.000,E1 311.472} C_DIS
LIN {X 0.032,Y -523.536,Z 1154.521,A 0.000,B 0.000,C 90.000,E1 309.725} C_DIS
LIN {X 0.050,Y -524.884,Z 1154.508,A 0.000,B 0.000,C 90.000,E1 307.397} C_DIS
LIN {X 0.193,Y -525.816,Z 1154.500,A 0.000,B 0.000,C 90.000,E1 305.931} C_DIS
LIN {X 0.127,Y -526.848,Z 1154.490,A 0.000,B 0.000,C 90.000,E1 304.199} C_DIS
LIN {X 0.149,Y -528.564,Z 1154.476,A 0.000,B 0.000,C 90.000,E1 301.592} C_DIS
LIN {X -0.009,Y -529.879,Z 1154.464,A 0.000,B 0.000,C 90.000,E1 299.589} C_DIS
LIN {X -0.189,Y -530.381,Z 1154.460,A 0.000,B 0.000,C 90.000,E1 298.743} C_DIS
LIN {X 0.235,Y -530.974,Z 1154.452,A 0.000,B 0.000,C 90.000,E1 297.257} C_DIS
LIN {X -0.046,Y -531.290,Z 1154.444,A 0.000,B 0.000,C 90.000,E1 295.848} C_DIS
LIN {X 0.155,Y -531.420,Z 1154.436,A 0.000,B 0.000,C 90.000,E1 294.387} C_DIS
LIN {X -0.162,Y -531.358,Z 1154.426,A 0.000,B 0.000,C 90.000,E1 292.695} C_DIS
LIN {X -0.195,Y -531.319,Z 1154.416,A 0.000,B 0.000,C 90.000,E1 290.972} C_DIS
LIN {X 0.075,Y -531.019,Z 1154.408,A 0.000,B 0.000,C 90.000,E1 289.504} C_DIS
LIN {X -0.022,Y -530.664,Z 1154.402,A 0.000,B 0.000,C 90.000,E1 288.362} C_DIS
LIN {X 0.084,Y -530.013,Z 1154.392,A 0.000,B 0.000,C 90.000,E1 286.622} C_DIS
LIN {X 0.029,Y -529.170,Z 1154.383,A 0.000,B 0.000,C 90.000,E1 284.898} C_DIS
LIN {X -0.080,Y -528.445,Z 1154.375,A 0.000,B 0.000,C 90.000,E1 283.467} C_DIS
LIN {X 0.032,Y -527.723,Z 1154.368,A 0.000,B 0.000,C 90.000,E1 282.299} C_DIS
LIN {X 0.191,Y -526.634,Z 1154.359,A 0.000,B 0.000,C 90.000,E1 280.546} C_DIS
LIN {X 0.249,Y -525.411,Z 1154.348,A 0.000,B 0.000,C 90.000,E1 278.511} C_DIS
LIN {X 0.183,Y -524.325,Z 1154.338,A 0.000,B 0.000,C 90.000,E1 276.777} C_DIS
LIN {X 0.035,Y -523.460,Z 1154.328,A 0.000,B 0.000,C 90.000,E1 275.049} C_DIS
LIN {X -0.125,Y -522.799,Z 1154.320,A 0.000,B 0.000,C 90.000,E1 273.612} C_DIS
LIN {X 0.150,Y -522.135,Z 1154.310,A 0.000,B 0.000,C 90.000,E1 271.835} C_DIS
LIN {X -0.066,Y -521.554,Z 1154.302,A 0.000,B 0.000,C 90.000,E1 270.401} C_DIS
LIN {X 0.165,Y -520.751,Z 1154.292,A 0.000,B 0.000,C 90.000,E1 268.625} C_DIS
LIN {X -0.078,Y -520.081,Z 1154.284,A 0.000,B 0.000,C 90.000,E1 267.192} C_DIS
LIN {X -0.219,Y -519.675,Z 1154.280,A 0.000,B 0.000,C 90.000,E1 266.331} C_DIS
LIN {X 0.154,Y -519.133,Z 1154.275,A 0.000,B 0.000,C 90.000,E1 265.412} C_DIS
LIN {X -0.020,Y -518.255,Z 1154.268,A 0.000,B 0.000,C 90.000,E1 264.261} C_DIS
LIN {X -0.225,Y -516.863,Z 1154.260,A 0.000,B 0.000,C 90.000,E1 262.818} C_DIS
LIN {X 0.031,Y -515.116,Z 1154.250,A 0.000,B 0.000,C 90.000,E1 261.027} C_DIS
LIN {X -0.094,Y -513.362,Z 1154.240,A 0.000,B 0.000,C 90.000,E1 259.275} C_DIS
LIN {X 0.253,Y -511.678,Z 1154.231,A 0.000,B 0.000,C 90.000,E1 257.465} C_DIS
LIN {X 0.165,Y -510.144,Z 1154.221,A 0.000,B 0.000,C 90.000,E1 255.700} C_DIS
LIN {X 0.164,Y -508.600,Z 1154.211,A 0.000,B 0.000,C 90.000,E1 253.921} C_DIS
LIN {X -0.217,Y -506.953,Z 1154.201,A 0.000,B 0.000,C 90.000,E1 252.181} C_DIS
LIN {X 0.002,Y -505.203,Z 1154.191,A 0.000,B 0.000,C 90.000,E1 250.369} C_DIS
LIN {X -0.209,Y -503.720,Z 1154.183,A 0.000,B 0.000,C 90.000,E1 248.901} C_DIS
LIN {X 0.204,Y -502.218,Z 1154.174,A 0.000,B 0.000,C 90.000,E1 247.358} C_DIS
LIN {X 0.118,Y -500.488,Z 1154.166,A 0.000,B 0.000,C 90.000,E1 245.869} C_DIS
LIN {X 0.138,Y -498.926,Z 1154.159,A 0.000,B 0.000,C 90.000,E1 244.665} C_DIS
LIN {X -0.036,Y -496.867,Z 1154.151,A 0.000,B 0.000,C 90.000,E1 243.179} C_DIS
LIN {X -0.112,Y -495.610,Z 1154.146,A 0.000,B 0.000,C 90.000,E1 242.281} C_DIS
LIN {X -0.079,Y -493.007,Z 1154.136,A 0.000,B 0.000,C 90.000,E1 240.461} C_DIS
LIN {X 0.034,Y -491.636,Z 1154.131,A 0.000,B 0.000,C 90.000,E1 239.537} C_DIS
LIN {X 0.209,Y -489.304,Z 1154.122,A 0.000,B 0.000,C 90.000,E1 237.995} C_DIS
LIN {X -0.184,Y -485.513,Z 1154.109,A 0.000,B 0.000,C 90.000,E1 235.595} C_DIS
LIN {X 0.224,Y -482.671,Z 1154.099,A 0.000,B 0.000,C 90.000,E1 233.703} C_DIS
LIN {X 0.165,Y -480.703,Z 1154.092,A 0.000,B 0.000,C 90.000,E1 232.477} C_DIS
LIN {X -0.017,Y -477.737,Z 1154.081,A 0.000,B 0.000,C 90.000,E1 230.642} C_DIS
LIN {X -0.179,Y -474.208,Z 1154.069,A 0.000,B 0.000,C 90.000,E1 228.485} C_DIS
LIN {X -0.166,Y -470.605,Z 1154.057,A 0.000,B 0.000,C 90.000,E1 226.296} C_DIS
LIN {X 0.233,Y -464.472,Z 1154.033,A 0.000,B 0.000,C 90.000,E1 221.838} C_DIS
LIN {X -0.174,Y -461.937,Z 1154.017,A 0.000,B 0.000,C 90.000,E1 219.036} C_DIS
LIN {X 0.106,Y -461.025,Z 1154.010,A 0.000,B 0.000,C 90.000,E1 217.729} C_DIS
LIN {X 0.081,Y -459.371,Z 1153.996,A 0.000,B 0.000,C 90.000,E1 215.185} C_DIS
LIN {X -0.070,Y -458.266,Z 1153.973,A 0.000,B 0.000,C 90.000,E1 211.052} C_DIS
LIN {X 0.062,Y -460.088,Z 1153.948,A 0.000,B 0.000,C 90.000,E1 206.565} C_DIS
LIN {X 0.112,Y -463.281,Z 1153.932,A 0.000,B 0.000,C 90.000,E1 203.695} C_DIS
LIN {X -0.082,Y -468.878,Z 1153.914,A 0.000,B 0.000,C 90.000,E1 200.556} C_DIS
LIN {X -0.111,Y -474.115,Z 1153.902,A 0.000,B 0.000,C 90.000,E1 198.362} C_DIS
LIN {X 0.145,Y -481.205,Z 1153.888,A 0.000,B 0.000,C 90.000,E1 195.843} C_DIS
LIN {X 0.017,Y -488.337,Z 1153.876,A 0.000,B 0.000,C 90.000,E1 193.703} C_DIS
LIN {X -0.067,Y -494.580,Z 1153.866,A 0.000,B 0.000,C 90.000,E1 191.883} C_DIS
LIN {X -0.112,Y -501.082,Z 1153.856,A 0.000,B 0.000,C 90.000,E1 190.074} C_DIS
LIN {X -0.038,Y -506.604,Z 1153.848,A 0.000,B 0.000,C 90.000,E1 188.568} C_DIS
LIN {X 0.076,Y -512.236,Z 1153.839,A 0.000,B 0.000,C 90.000,E1 187.068} C_DIS
LIN {X -0.211,Y -517.785,Z 1153.831,A 0.000,B 0.000,C 90.000,E1 185.625} C_DIS
LIN {X 0.069,Y -523.280,Z 1153.823,A 0.000,B 0.000,C 90.000,E1 184.131} C_DIS
LIN {X -0.075,Y -528.728,Z 1153.815,A 0.000,B 0.000,C 90.000,E1 182.694} C_DIS
LIN {X -0.155,Y -534.154,Z 1153.807,A 0.000,B 0.000,C 90.000,E1 181.260} C_DIS
LIN {X -0.147,Y -539.541,Z 1153.799,A 0.000,B 0.000,C 90.000,E1 179.828} C_DIS
LIN {X -0.042,Y -545.029,Z 1153.791,A 0.000,B 0.000,C 90.000,E1 178.396} C_DIS
LIN {X -0.188,Y -553.719,Z 1153.779,A 0.000,B 0.000,C 90.000,E1 176.159} C_DIS
LIN {X 0.152,Y -558.073,Z 1153.772,A 0.000,B 0.000,C 90.000,E1 175.008} C_DIS
LIN {X 0.237,Y -564.499,Z 1153.763,A 0.000,B 0.000,C 90.000,E1 173.337} C_DIS
LIN {X -0.213,Y -569.862,Z 1153.755,A 0.000,B 0.000,C 90.000,E1 172.008} C_DIS
LIN {X 0.187,Y -576.194,Z 1153.746,A 0.000,B 0.000,C 90.000,E1 170.330} C_DIS
LIN {X 0.241,Y -582.439,Z 1153.737,A 0.000,B 0.000,C 90.000,E1 168.701} C_DIS
LIN {X -0.198,Y -585.530,Z 1153.733,A 0.000,B 0.000,C 90.000,E1 167.937} C_DIS
LIN {X 0.222,Y -589.509,Z 1153.727,A 0.000,B 0.000,C 90.000,E1 166.825} C_DIS
LIN {X 0.263,Y -593.368,Z 1153.721,A 0.000,B 0.000,C 90.000,E1 165.755} C_DIS
LIN {X 0.074,Y -597.958,Z 1153.714,A 0.000,B 0.000,C 90.000,E1 164.448} C_DIS
LIN {X 0.242,Y -601.515,Z 1153.708,A 0.000,B 0.000,C 90.000,E1 163.378} C_DIS
LIN {X -0.124,Y -604.943,Z 1153.702,A 0.000,B 0.000,C 90.000,E1 162.362} C_DIS
LIN {X 0.046,Y -609.023,Z 1153.695,A 0.000,B 0.000,C 90.000,E1 161.040} C_DIS
LIN {X -0.352,Y -613.631,Z 1153.686,A 0.000,B 0.000,C 90.000,E1 159.518} C_DIS
LIN {X -0.155,Y -616.569,Z 1153.680,A 0.000,B 0.000,C 90.000,E1 158.465} C_DIS
LIN {X -0.181,Y -620.802,Z 1153.672,A 0.000,B 0.000,C 90.000,E1 156.922} C_DIS
LIN {X 0.116,Y -623.506,Z 1153.666,A 0.000,B 0.000,C 90.000,E1 155.869} C_DIS
LIN {X 0.166,Y -627.480,Z 1153.658,A 0.000,B 0.000,C 90.000,E1 154.332} C_DIS
LIN {X -0.006,Y -630.600,Z 1153.651,A 0.000,B 0.000,C 90.000,E1 153.076} C_DIS
LIN {X -0.114,Y -633.665,Z 1153.643,A 0.000,B 0.000,C 90.000,E1 151.820} C_DIS
LIN {X 0.089,Y -636.545,Z 1153.636,A 0.000,B 0.000,C 90.000,E1 150.539} C_DIS
LIN {X -0.010,Y -638.165,Z 1153.632,A 0.000,B 0.000,C 90.000,E1 149.793} C_DIS
LIN {X -0.033,Y -640.314,Z 1153.627,A 0.000,B 0.000,C 90.000,E1 148.791} C_DIS
LIN {X 0.024,Y -642.754,Z 1153.620,A 0.000,B 0.000,C 90.000,E1 147.533} C_DIS
LIN {X -0.082,Y -645.027,Z 1153.613,A 0.000,B 0.000,C 90.000,E1 146.294} C_DIS
LIN {X -0.152,Y -647.240,Z 1153.606,A 0.000,B 0.000,C 90.000,E1 145.055} C_DIS
LIN {X 0.185,Y -649.389,Z 1153.599,A 0.000,B 0.000,C 90.000,E1 143.783} C_DIS
LIN {X 0.010,Y -652.238,Z 1153.589,A 0.000,B 0.000,C 90.000,E1 142.065} C_DIS
LIN {X 0.247,Y -655.784,Z 1153.578,A 0.000,B 0.000,C 90.000,E1 140.070} C_DIS
LIN {X 0.150,Y -657.765,Z 1153.573,A 0.000,B 0.000,C 90.000,E1 139.094} C_DIS
LIN {X 0.021,Y -660.762,Z 1153.565,A 0.000,B 0.000,C 90.000,E1 137.634} C_DIS
LIN {X 0.399,Y -663.670,Z 1153.557,A 0.000,B 0.000,C 90.000,E1 136.134} C_DIS
LIN {X -0.083,Y -669.437,Z 1153.542,A 0.000,B 0.000,C 90.000,E1 133.500} C_DIS
LIN {X 0.066,Y -673.946,Z 1153.531,A 0.000,B 0.000,C 90.000,E1 131.553} C_DIS
LIN {X 0.020,Y -679.825,Z 1153.518,A 0.000,B 0.000,C 90.000,E1 129.152} C_DIS
LIN {X -0.151,Y -682.876,Z 1153.511,A 0.000,B 0.000,C 90.000,E1 127.971} C_DIS
LIN {X -0.455,Y -687.639,Z 1153.500,A 0.000,B 0.000,C 90.000,E1 126.091} C_DIS
LIN {X 0.224,Y -691.131,Z 1153.492,A 0.000,B 0.000,C 90.000,E1 124.612} C_DIS
LIN {X -0.026,Y -693.970,Z 1153.486,A 0.000,B 0.000,C 90.000,E1 123.452} C_DIS
LIN {X 0.118,Y -696.148,Z 1153.481,A 0.000,B 0.000,C 90.000,E1 122.498} C_DIS
LIN {X -0.305,Y -698.108,Z 1153.475,A 0.000,B 0.000,C 90.000,E1 121.592} C_DIS
LIN {X 0.122,Y -699.845,Z 1153.470,A 0.000,B 0.000,C 90.000,E1 120.620} C_DIS
LIN {X -0.078,Y -702.799,Z 1153.461,A 0.000,B 0.000,C 90.000,E1 118.999} C_DIS
LIN {X 0.091,Y -704.430,Z 1153.456,A 0.000,B 0.000,C 90.000,E1 118.052} C_DIS
LIN {X -0.296,Y -705.398,Z 1153.452,A 0.000,B 0.000,C 90.000,E1 117.385} C_DIS
LIN {X 0.285,Y -705.893,Z 1153.449,A 0.000,B 0.000,C 90.000,E1 116.873} C_DIS
LIN {X 0.169,Y -706.505,Z 1153.443,A 0.000,B 0.000,C 90.000,E1 115.720} C_DIS
LIN {X 0.109,Y -706.537,Z 1153.439,A 0.000,B 0.000,C 90.000,E1 115.027} C_DIS
LIN {X -0.242,Y -706.414,Z 1153.437,A 0.000,B 0.000,C 90.000,E1 114.591} C_DIS
LIN {X 0.343,Y -705.525,Z 1153.434,A 0.000,B 0.000,C 90.000,E1 114.079} C_DIS
LIN {X -0.299,Y -704.966,Z 1153.433,A 0.000,B 0.000,C 90.000,E1 113.898} C_DIS
LIN {X 0.134,Y -702.390,Z 1153.429,A 0.000,B 0.000,C 90.000,E1 113.281} C_DIS
LIN {X -0.370,Y -701.526,Z 1153.429,A 0.000,B 0.000,C 90.000,E1 113.206} C_DIS
LIN {X -0.102,Y -697.095,Z 1153.426,A 0.000,B 0.000,C 90.000,E1 112.717} C_DIS
LIN {X 0.027,Y -695.509,Z 1153.426,A 0.000,B 0.000,C 90.000,E1 112.589} C_DIS
LIN {X 0.155,Y -692.680,Z 1153.425,A 0.000,B 0.000,C 90.000,E1 112.461} C_DIS
LIN {X 0.014,Y -686.804,Z 1153.424,A 0.000,B 0.000,C 90.000,E1 112.280} C_DIS
LIN {X 0.238,Y -684.581,Z 1153.424,A 0.000,B 0.000,C 90.000,E1 112.206} C_DIS
LIN {X 0.131,Y -676.718,Z 1153.423,A 0.000,B 0.000,C 90.000,E1 112.153} C_DIS
LIN {X 0.069,Y -603.805,Z 1153.423,A 0.000,B 0.000,C 90.000,E1 112.153} C_DIS
LIN {X -0.097,Y -600.471,Z 1153.422,A 0.000,B 0.000,C 90.000,E1 111.950} C_DIS
LIN {X 0.153,Y -591.780,Z 1153.418,A 0.000,B 0.000,C 90.000,E1 111.227} C_DIS
LIN {X -0.152,Y -578.176,Z 1153.411,A 0.000,B 0.000,C 90.000,E1 110.066} C_DIS
LIN {X 0.054,Y -573.943,Z 1153.409,A 0.000,B 0.000,C 90.000,E1 109.685} C_DIS
LIN {X 0.221,Y -567.940,Z 1153.407,A 0.000,B 0.000,C 90.000,E1 109.214} C_DIS
LIN {X -0.142,Y -560.015,Z 1153.404,A 0.000,B 0.000,C 90.000,E1 108.725} C_DIS
LIN {X -0.078,Y -555.330,Z 1153.402,A 0.000,B 0.000,C 90.000,E1 108.417} C_DIS
LIN {X -0.060,Y -551.535,Z 1153.401,A 0.000,B 0.000,C 90.000,E1 108.109} C_DIS
LIN {X 0.090,Y -550.175,Z 1153.399,A 0.000,B 0.000,C 90.000,E1 107.873} C_DIS
LIN {X 0.048,Y -550.164,Z 1153.399,A 0.000,B 0.000,C 90.000,E1 107.873} C_DIS
LIN {X 0.264,Y -549.856,Z 1153.397,A 0.000,B 0.000,C 90.000,E1 107.457} C_DIS
LIN {X -0.046,Y -551.073,Z 1153.387,A 0.000,B 0.000,C 90.000,E1 105.607} C_DIS
LIN {X -0.169,Y -552.422,Z 1153.377,A 0.000,B 0.000,C 90.000,E1 103.939} C_DIS
LIN {X -0.114,Y -553.637,Z 1153.370,A 0.000,B 0.000,C 90.000,E1 102.535} C_DIS
LIN {X 0.101,Y -555.236,Z 1153.360,A 0.000,B 0.000,C 90.000,E1 100.838} C_DIS
LIN {X 0.249,Y -556.811,Z 1153.351,A 0.000,B 0.000,C 90.000,E1 99.151} C_DIS
LIN {X -0.072,Y -558.470,Z 1153.340,A 0.000,B 0.000,C 90.000,E1 97.239} C_DIS
LIN {X 0.122,Y -559.916,Z 1153.329,A 0.000,B 0.000,C 90.000,E1 95.277} C_DIS
LIN {X -0.055,Y -560.776,Z 1153.323,A 0.000,B 0.000,C 90.000,E1 94.188} C_DIS
LIN {X 0.106,Y -562.235,Z 1153.313,A 0.000,B 0.000,C 90.000,E1 92.236} C_DIS
LIN {X 0.066,Y -563.316,Z 1153.305,A 0.000,B 0.000,C 90.000,E1 90.859} C_DIS
LIN {X 0.140,Y -564.463,Z 1153.296,A 0.000,B 0.000,C 90.000,E1 89.198} C_DIS
LIN {X 0.029,Y -565.154,Z 1153.290,A 0.000,B 0.000,C 90.000,E1 88.108} C_DIS
LIN {X 0.155,Y -566.110,Z 1153.280,A 0.000,B 0.000,C 90.000,E1 86.445} C_DIS
LIN {X -0.078,Y -567.220,Z 1153.270,A 0.000,B 0.000,C 90.000,E1 84.546} C_DIS
LIN {X -0.266,Y -567.725,Z 1153.265,A 0.000,B 0.000,C 90.000,E1 83.742} C_DIS
LIN {X 0.061,Y -568.628,Z 1153.256,A 0.000,B 0.000,C 90.000,E1 82.064} C_DIS
LIN {X 0.044,Y -569.167,Z 1153.250,A 0.000,B 0.000,C 90.000,E1 80.971} C_DIS
LIN {X -0.264,Y -569.806,Z 1153.242,A 0.000,B 0.000,C 90.000,E1 79.634} C_DIS
LIN {X 0.108,Y -570.465,Z 1153.235,A 0.000,B 0.000,C 90.000,E1 78.229} C_DIS
LIN {X -0.243,Y -571.395,Z 1153.224,A 0.000,B 0.000,C 90.000,E1 76.353} C_DIS
LIN {X 0.257,Y -572.352,Z 1153.214,A 0.000,B 0.000,C 90.000,E1 74.393} C_DIS
LIN {X 0.038,Y -573.628,Z 1153.201,A 0.000,B 0.000,C 90.000,E1 72.236} C_DIS
LIN {X 0.204,Y -574.975,Z 1153.191,A 0.000,B 0.000,C 90.000,E1 70.315} C_DIS
LIN {X -0.132,Y -576.301,Z 1153.182,A 0.000,B 0.000,C 90.000,E1 68.720} C_DIS
LIN {X -0.069,Y -577.581,Z 1153.174,A 0.000,B 0.000,C 90.000,E1 67.358} C_DIS
LIN {X -0.134,Y -578.678,Z 1153.168,A 0.000,B 0.000,C 90.000,E1 66.282} C_DIS
LIN {X -0.315,Y -580.380,Z 1153.158,A 0.000,B 0.000,C 90.000,E1 64.409} C_DIS
LIN {X -0.083,Y -581.390,Z 1153.152,A 0.000,B 0.000,C 90.000,E1 63.307} C_DIS
LIN {X -0.087,Y -582.820,Z 1153.143,A 0.000,B 0.000,C 90.000,E1 61.691} C_DIS
LIN {X 0.055,Y -583.962,Z 1153.135,A 0.000,B 0.000,C 90.000,E1 60.333} C_DIS
LIN {X -0.136,Y -585.213,Z 1153.126,A 0.000,B 0.000,C 90.000,E1 58.742} C_DIS
LIN {X -0.001,Y -586.252,Z 1153.117,A 0.000,B 0.000,C 90.000,E1 57.120} C_DIS
LIN {X -0.201,Y -587.087,Z 1153.110,A 0.000,B 0.000,C 90.000,E1 55.801} C_DIS
LIN {X -0.190,Y -588.083,Z 1153.101,A 0.000,B 0.000,C 90.000,E1 54.196} C_DIS
LIN {X -0.081,Y -589.120,Z 1153.091,A 0.000,B 0.000,C 90.000,E1 52.316} C_DIS
LIN {X 0.104,Y -589.842,Z 1153.083,A 0.000,B 0.000,C 90.000,E1 50.964} C_DIS
LIN {X 0.203,Y -590.360,Z 1153.076,A 0.000,B 0.000,C 90.000,E1 49.622} C_DIS
LIN {X -0.137,Y -590.648,Z 1153.068,A 0.000,B 0.000,C 90.000,E1 48.324} C_DIS
LIN {X 0.167,Y -590.728,Z 1153.063,A 0.000,B 0.000,C 90.000,E1 47.229} C_DIS
LIN {X 0.235,Y -590.650,Z 1153.055,A 0.000,B 0.000,C 90.000,E1 45.891} C_DIS
LIN {X 0.115,Y -590.462,Z 1153.049,A 0.000,B 0.000,C 90.000,E1 44.838} C_DIS
LIN {X 0.231,Y -590.165,Z 1153.045,A 0.000,B 0.000,C 90.000,E1 44.028} C_DIS
LIN {X 0.097,Y -589.518,Z 1153.039,A 0.000,B 0.000,C 90.000,E1 42.975} C_DIS
LIN {X -0.015,Y -588.776,Z 1153.033,A 0.000,B 0.000,C 90.000,E1 41.919} C_DIS
LIN {X -0.129,Y -587.699,Z 1153.027,A 0.000,B 0.000,C 90.000,E1 40.862} C_DIS
LIN {X -0.190,Y -587.165,Z 1153.024,A 0.000,B 0.000,C 90.000,E1 40.334} C_DIS
LIN {X 0.052,Y -585.142,Z 1153.015,A 0.000,B 0.000,C 90.000,E1 38.705} C_DIS
LIN {X -0.030,Y -584.432,Z 1153.012,A 0.000,B 0.000,C 90.000,E1 38.177} C_DIS
LIN {X 0.071,Y -582.187,Z 1153.005,A 0.000,B 0.000,C 90.000,E1 36.824} C_DIS
LIN {X 0.132,Y -580.522,Z 1153.000,A 0.000,B 0.000,C 90.000,E1 36.011} C_DIS
LIN {X 0.134,Y -579.351,Z 1152.997,A 0.000,B 0.000,C 90.000,E1 35.471} C_DIS
LIN {X -0.177,Y -577.282,Z 1152.993,A 0.000,B 0.000,C 90.000,E1 34.692} C_DIS
LIN {X -0.035,Y -574.935,Z 1152.988,A 0.000,B 0.000,C 90.000,E1 33.865} C_DIS
LIN {X 0.256,Y -573.180,Z 1152.985,A 0.000,B 0.000,C 90.000,E1 33.293} C_DIS
LIN {X 0.041,Y -570.194,Z 1152.981,A 0.000,B 0.000,C 90.000,E1 32.498} C_DIS
LIN {X 0.104,Y -566.958,Z 1152.976,A 0.000,B 0.000,C 90.000,E1 31.671} C_DIS
LIN {X -0.080,Y -561.882,Z 1152.970,A 0.000,B 0.000,C 90.000,E1 30.590} C_DIS
LIN {X 0.076,Y -557.618,Z 1152.965,A 0.000,B 0.000,C 90.000,E1 29.745} C_DIS
LIN {X -0.076,Y -554.590,Z 1152.962,A 0.000,B 0.000,C 90.000,E1 29.205} C_DIS
LIN {X 0.119,Y -550.529,Z 1152.958,A 0.000,B 0.000,C 90.000,E1 28.487} C_DIS
LIN {X -0.227,Y -547.960,Z 1152.956,A 0.000,B 0.000,C 90.000,E1 28.103} C_DIS
